LIN {X 0,Y 267.437,Z 177.913,A -85,B 0,C 180,E1 11882.304,E2 11882.304} C_VEL
LIN {X 0,Y 262.666,Z 169.182,A -85,B 0,C 180,E1 11878.91,E2 11878.91} C_VEL
LIN {X 0,Y 261.698,Z 164.317,A -85,B 0,C 180,E1 11875.398,E2 11875.398} C_VEL
LIN {X 0,Y 260.906,Z 160.303,A -85,B 0,C 180,E1 11871.391,E2 11871.391} C_VEL
LIN {X 0,Y 260.574,Z 157.948,A -85,B 0,C 180,E1 11867.817,E2 11867.817} C_VEL
LIN {X 0,Y 260.431,Z 157.03,A -85,B 0,C 180,E1 11862.806,E2 11862.806} C_VEL
LIN {X 0,Y 260.984,Z 157.956,A -85,B 0,C 180,E1 11858.587,E2 11858.587} C_VEL
LIN {X 0,Y 261.9,Z 159.655,A -85,B 0,C 180,E1 11855.41,E2 11855.41} C_VEL
LIN {X 0,Y 263.162,Z 163.319,A -85,B 0,C 180,E1 11851.646,E2 11851.646} C_VEL
LIN {X 0,Y 264.344,Z 166.629,A -85,B 0,C 180,E1 11849.225,E2 11849.225} C_VEL
LIN {X 0,Y 269.556,Z 174.246,A -85,B 0,C 180,E1 11846.002,E2 11846.002} C_VEL
LIN {X 0,Y 274.151,Z 181.59,A -85,B 0,C 180,E1 11843.655,E2 11843.655} C_VEL
LIN {X 0,Y 279.034,Z 190.083,A -85,B 0,C 180,E1 11841.462,E2 11841.462} C_VEL
LIN {X 0,Y 281.087,Z 194.443,A -85,B 0,C 180,E1 11840.571,E2 11840.571} C_VEL
LIN {X 0,Y 281.207,Z 206.246,A -85,B 0,C 180,E1 11839.931,E2 11839.931} C_VEL
LIN {X 0,Y 271.188,Z 340.936,A -85,B 0,C 180,E1 11836.322,E2 11836.322} C_VEL
LIN {X 0,Y 268.525,Z 359.447,A -85,B 0,C 180,E1 11835.523,E2 11835.523} C_VEL
LIN {X 0,Y 264.865,Z 376.74,A -85,B 0,C 180,E1 11834.449,E2 11834.449} C_VEL
LIN {X 0,Y 260.399,Z 393.338,A -85,B 0,C 180,E1 11833.028,E2 11833.028} C_VEL
LIN {X 0,Y 255.563,Z 408.467,A -85,B 0,C 180,E1 11831.308,E2 11831.308} C_VEL
LIN {X 0,Y 250.235,Z 423.172,A -85,B 0,C 180,E1 11829.149,E2 11829.149} C_VEL
LIN {X 0,Y 244.431,Z 437.876,A -85,B 0,C 180,E1 11826.381,E2 11826.381} C_VEL
LIN {X 0,Y 238.982,Z 450.923,A -85,B 0,C 180,E1 11823.237,E2 11823.237} C_VEL
LIN {X 0,Y 234.103,Z 462.435,A -85,B 0,C 180,E1 11819.7,E2 11819.7} C_VEL
LIN {X 0,Y 230.027,Z 472.48,A -85,B 0,C 180,E1 11815.766,E2 11815.766} C_VEL
LIN {X 0,Y 226.993,Z 481.069,A -85,B 0,C 180,E1 11811.446,E2 11811.446} C_VEL
LIN {X 0,Y 225.186,Z 488.132,A -85,B 0,C 180,E1 11806.776,E2 11806.776} C_VEL
LIN {X 0,Y 224.728,Z 493.306,A -85,B 0,C 180,E1 11802.072,E2 11802.072} C_VEL
LIN {X 0,Y 225.341,Z 496.657,A -85,B 0,C 180,E1 11797.395,E2 11797.395} C_VEL
LIN {X 0,Y 226.348,Z 498.067,A -85,B 0,C 180,E1 11793.294,E2 11793.294} C_VEL
LIN {X 0,Y 226.857,Z 498.055,A -85,B 0,C 180,E1 11790.002,E2 11790.002} C_VEL
LIN {X 0,Y 226.415,Z 496.907,A -85,B 0,C 180,E1 11786.394,E2 11786.394} C_VEL
LIN {X 0,Y 225.507,Z 494.955,A -85,B 0,C 180,E1 11782.614,E2 11782.614} C_VEL
LIN {X 0,Y 224.98,Z 491.385,A -85,B 0,C 180,E1 11778.985,E2 11778.985} C_VEL
LIN {X 0,Y 225.066,Z 485.569,A -85,B 0,C 180,E1 11775.071,E2 11775.071} C_VEL
LIN {X 0,Y 225.901,Z 477.705,A -85,B 0,C 180,E1 11771.294,E2 11771.294} C_VEL
LIN {X 0,Y 228.497,Z 464.106,A -85,B 0,C 180,E1 11765.989,E2 11765.989} C_VEL
LIN {X 0,Y 231.379,Z 452.377,A -85,B 0,C 180,E1 11762.358,E2 11762.358} C_VEL
LIN {X 0,Y 234.793,Z 439.326,A -85,B 0,C 180,E1 11759.129,E2 11759.129} C_VEL
LIN {X 0,Y 238.397,Z 425.351,A -85,B 0,C 180,E1 11756.387,E2 11756.387} C_VEL
LIN {X 0,Y 242.028,Z 410.421,A -85,B 0,C 180,E1 11754.067,E2 11754.067} C_VEL
LIN {X 0,Y 245.616,Z 393.93,A -85,B 0,C 180,E1 11752.073,E2 11752.073} C_VEL
LIN {X 0,Y 248.682,Z 377.423,A -85,B 0,C 180,E1 11750.564,E2 11750.564} C_VEL
LIN {X 0,Y 251.306,Z 359.444,A -85,B 0,C 180,E1 11749.376,E2 11749.376} C_VEL
LIN {X 0,Y 252.921,Z 341.212,A -85,B 0,C 180,E1 11748.58,E2 11748.58} C_VEL
LIN {X 0,Y 260.465,Z 182.567,A -85,B 0,C 180,E1 11744.28,E2 11744.28} C_VEL
LIN {X 0,Y 260.223,Z 166.645,A -85,B 0,C 180,E1 11743.682,E2 11743.682} C_VEL
LIN {X 0,Y 256.691,Z 159.312,A -85,B 0,C 180,E1 11742.821,E2 11742.821} C_VEL
LIN {X 0,Y 249.435,Z 140.807,A -85,B 0,C 180,E1 11739.148,E2 11739.148} C_VEL
LIN {X 0,Y 242.573,Z 125.136,A -85,B 0,C 180,E1 11735.534,E2 11735.534} C_VEL
LIN {X 0,Y 235.678,Z 110.896,A -85,B 0,C 180,E1 11731.74,E2 11731.74} C_VEL
LIN {X 0,Y 230.937,Z 101.989,A -85,B 0,C 180,E1 11729.006,E2 11729.006} C_VEL
LIN {X 0,Y 229.132,Z 98.21,A -85,B 0,C 180,E1 11727.834,E2 11727.834} C_VEL
LIN {X 0,Y 227.177,Z 95.014,A -85,B 0,C 180,E1 11726.674,E2 11726.674} C_VEL
LIN {X 0,Y 226.869,Z 93.749,A -85,B 0,C 180,E1 11726.149,E2 11726.149} C_VEL
LIN {X 0,Y 226.849,Z 93.536,A -85,B 0,C 180,E1 11720.875,E2 11720.875} C_VEL
LIN {X 0,Y 226.834,Z 93.529,A -85,B 0,C 180,E1 11715.597,E2 11715.597} C_VEL
LIN {X 0,Y 226.832,Z 93.525,A -85,B 0,C 180,E1 11710.411,E2 11710.411} C_VEL
LIN {X 0,Y 226.837,Z 93.521,A -85,B 0,C 180,E1 11705.311,E2 11705.311} C_VEL
LIN {X 0,Y 226.825,Z 93.521,A -85,B 0,C 180,E1 11699.999,E2 11699.999} C_VEL
LIN {X 0,Y 226.83,Z 93.523,A -85,B 0,C 180,E1 11694.942,E2 11694.942} C_VEL
LIN {X 0,Y 226.833,Z 93.526,A -85,B 0,C 180,E1 11689.587,E2 11689.587} C_VEL
LIN {X 0,Y 226.866,Z 93.724,A -85,B 0,C 180,E1 11685.711,E2 11685.711} C_VEL
LIN {X 0,Y 227.21,Z 95.191,A -85,B 0,C 180,E1 11684.69,E2 11684.69} C_VEL
LIN {X 0,Y 229.356,Z 98.44,A -85,B 0,C 180,E1 11682.494,E2 11682.494} C_VEL
LIN {X 0,Y 230.666,Z 99.715,A -85,B 0,C 180,E1 11681.421,E2 11681.421} C_VEL
LIN {X 0,Y 232.401,Z 103.285,A -85,B 0,C 180,E1 11679.605,E2 11679.605} C_VEL
LIN {X 0,Y 233.957,Z 105.019,A -85,B 0,C 180,E1 11678.436,E2 11678.436} C_VEL
LIN {X 0,Y 236.12,Z 109.062,A -85,B 0,C 180,E1 11676.543,E2 11676.543} C_VEL
LIN {X 0,Y 237.292,Z 111.038,A -85,B 0,C 180,E1 11675.61,E2 11675.61} C_VEL
LIN {X 0,Y 240.213,Z 116.403,A -85,B 0,C 180,E1 11673.285,E2 11673.285} C_VEL
LIN {X 0,Y 243.943,Z 123.406,A -85,B 0,C 180,E1 11670.537,E2 11670.537} C_VEL
LIN {X 0,Y 248.961,Z 134.345,A -85,B 0,C 180,E1 11666.893,E2 11666.893} C_VEL
LIN {X 0,Y 253.489,Z 146.18,A -85,B 0,C 180,E1 11663.444,E2 11663.444} C_VEL
LIN {X 0,Y 257.748,Z 159.766,A -85,B 0,C 180,E1 11660.057,E2 11660.057} C_VEL
LIN {X 0,Y 259.774,Z 168.609,A -85,B 0,C 180,E1 11658.136,E2 11658.136} C_VEL
LIN {X 0,Y 256.196,Z 205.517,A -85,B 0,C 180,E1 11653.073,E2 11653.073} C_VEL
LIN {X 0,Y 255.073,Z 219.925,A -85,B 0,C 180,E1 11651.192,E2 11651.192} C_VEL
LIN {X 0,Y 255.745,Z 226.346,A -85,B 0,C 180,E1 11650.844,E2 11650.844} C_VEL
LIN {X 0,Y 251.79,Z 315.486,A -85,B 0,C 180,E1 11648.415,E2 11648.415} C_VEL
LIN {X 0,Y 251.344,Z 337.034,A -85,B 0,C 180,E1 11647.632,E2 11647.632} C_VEL
LIN {X 0,Y 250.337,Z 351.44,A -85,B 0,C 180,E1 11646.724,E2 11646.724} C_VEL
LIN {X 0,Y 248.542,Z 365.675,A -85,B 0,C 180,E1 11645.398,E2 11645.398} C_VEL
LIN {X 0,Y 246.267,Z 378.333,A -85,B 0,C 180,E1 11643.793,E2 11643.793} C_VEL
LIN {X 0,Y 243.611,Z 390.139,A -85,B 0,C 180,E1 11641.831,E2 11641.831} C_VEL
LIN {X 0,Y 240.515,Z 401.442,A -85,B 0,C 180,E1 11639.374,E2 11639.374} C_VEL
LIN {X 0,Y 237.305,Z 411.378,A -85,B 0,C 180,E1 11636.524,E2 11636.524} C_VEL
LIN {X 0,Y 234.397,Z 419.352,A -85,B 0,C 180,E1 11633.49,E2 11633.49} C_VEL
LIN {X 0,Y 231.822,Z 425.764,A -85,B 0,C 180,E1 11630.182,E2 11630.182} C_VEL
LIN {X 0,Y 229.746,Z 430.445,A -85,B 0,C 180,E1 11626.69,E2 11626.69} C_VEL
LIN {X 0,Y 228.185,Z 433.478,A -85,B 0,C 180,E1 11622.911,E2 11622.911} C_VEL
LIN {X 0,Y 227.257,Z 434.673,A -85,B 0,C 180,E1 11619.111,E2 11619.111} C_VEL
LIN {X 0,Y 226.912,Z 434.059,A -85,B 0,C 180,E1 11615.219,E2 11615.219} C_VEL
LIN {X 0,Y 227.15,Z 431.504,A -85,B 0,C 180,E1 11611.259,E2 11611.259} C_VEL
LIN {X 0,Y 227.948,Z 427.101,A -85,B 0,C 180,E1 11607.484,E2 11607.484} C_VEL
LIN {X 0,Y 229.216,Z 421.057,A -85,B 0,C 180,E1 11603.989,E2 11603.989} C_VEL
LIN {X 0,Y 230.876,Z 413.508,A -85,B 0,C 180,E1 11600.778,E2 11600.778} C_VEL
LIN {X 0,Y 232.823,Z 404.48,A -85,B 0,C 180,E1 11597.851,E2 11597.851} C_VEL
LIN {X 0,Y 235.023,Z 393.302,A -85,B 0,C 180,E1 11595.083,E2 11595.083} C_VEL
LIN {X 0,Y 236.437,Z 385.836,A -85,B 0,C 180,E1 11593.539,E2 11593.539} C_VEL
LIN {X 0,Y 237.322,Z 385.675,A -85,B 0,C 180,E1 11593.098,E2 11593.098} C_VEL
LIN {X 0,Y 237.457,Z 386.342,A -85,B 0,C 180,E1 11592.909,E2 11592.909} C_VEL
LIN {X 0,Y 234.65,Z 398.324,A -85,B 0,C 180,E1 11590.068,E2 11590.068} C_VEL
LIN {X 0,Y 232.114,Z 408.776,A -85,B 0,C 180,E1 11586.92,E2 11586.92} C_VEL
LIN {X 0,Y 229.927,Z 417.813,A -85,B 0,C 180,E1 11583.389,E2 11583.389} C_VEL
LIN {X 0,Y 228.359,Z 424.842,A -85,B 0,C 180,E1 11579.765,E2 11579.765} C_VEL
LIN {X 0,Y 227.33,Z 430.447,A -85,B 0,C 180,E1 11575.736,E2 11575.736} C_VEL
LIN {X 0,Y 226.986,Z 433.918,A -85,B 0,C 180,E1 11571.923,E2 11571.923} C_VEL
LIN {X 0,Y 227.285,Z 435.822,A -85,B 0,C 180,E1 11567.694,E2 11567.694} C_VEL
LIN {X 0,Y 228.271,Z 435.874,A -85,B 0,C 180,E1 11563.719,E2 11563.719} C_VEL
LIN {X 0,Y 230.027,Z 434.082,A -85,B 0,C 180,E1 11559.701,E2 11559.701} C_VEL
LIN {X 0,Y 232.613,Z 430.513,A -85,B 0,C 180,E1 11555.774,E2 11555.774} C_VEL
LIN {X 0,Y 235.937,Z 425.091,A -85,B 0,C 180,E1 11552.05,E2 11552.05} C_VEL
LIN {X 0,Y 240.029,Z 417.755,A -85,B 0,C 180,E1 11548.484,E2 11548.484} C_VEL
LIN {X 0,Y 244.454,Z 408.927,A -85,B 0,C 180,E1 11545.319,E2 11545.319} C_VEL
LIN {X 0,Y 249.258,Z 398.306,A -85,B 0,C 180,E1 11542.401,E2 11542.401} C_VEL
LIN {X 0,Y 253.856,Z 386.726,A -85,B 0,C 180,E1 11539.953,E2 11539.953} C_VEL
LIN {X 0,Y 258.341,Z 373.716,A -85,B 0,C 180,E1 11537.804,E2 11537.804} C_VEL
LIN {X 0,Y 262.44,Z 359.675,A -85,B 0,C 180,E1 11535.998,E2 11535.998} C_VEL
LIN {X 0,Y 266.113,Z 344.035,A -85,B 0,C 180,E1 11534.47,E2 11534.47} C_VEL
LIN {X 0,Y 268.945,Z 328.005,A -85,B 0,C 180,E1 11533.321,E2 11533.321} C_VEL
LIN {X 0,Y 271.021,Z 310.302,A -85,B 0,C 180,E1 11532.464,E2 11532.464} C_VEL
LIN {X 0,Y 273.763,Z 280.354,A -85,B 0,C 180,E1 11531.473,E2 11531.473} C_VEL
LIN {X 0,Y 273.908,Z 272.836,A -85,B 0,C 180,E1 11531.068,E2 11531.068} C_VEL
LIN {X 0,Y 272.225,Z 253.256,A -85,B 0,C 180,E1 11529.371,E2 11529.371} C_VEL
LIN {X 0,Y 272.444,Z 246.79,A -85,B 0,C 180,E1 11529.038,E2 11529.038} C_VEL
LIN {X 0,Y 273.723,Z 232.593,A -85,B 0,C 180,E1 11528.561,E2 11528.561} C_VEL
LIN {X 0,Y 272.08,Z 208.308,A -85,B 0,C 180,E1 11526.436,E2 11526.436} C_VEL
LIN {X 0,Y 271.119,Z 198.139,A -85,B 0,C 180,E1 11525.371,E2 11525.371} C_VEL
LIN {X 0,Y 267.119,Z 189.254,A -85,B 0,C 180,E1 11523.058,E2 11523.058} C_VEL
LIN {X 0,Y 263.16,Z 181.691,A -85,B 0,C 180,E1 11520.49,E2 11520.49} C_VEL
LIN {X 0,Y 259.632,Z 175.218,A -85,B 0,C 180,E1 11517.738,E2 11517.738} C_VEL
LIN {X 0,Y 256.045,Z 168.731,A -85,B 0,C 180,E1 11513.948,E2 11513.948} C_VEL
LIN {X 0,Y 255.481,Z 165.908,A -85,B 0,C 180,E1 11510.767,E2 11510.767} C_VEL
LIN {X 0,Y 255.299,Z 163.935,A -85,B 0,C 180,E1 11507.561,E2 11507.561} C_VEL
LIN {X 0,Y 255.269,Z 163.135,A -85,B 0,C 180,E1 11502.682,E2 11502.682} C_VEL
LIN {X 0,Y 255.846,Z 164.125,A -85,B 0,C 180,E1 11498.448,E2 11498.448} C_VEL
LIN {X 0,Y 256.662,Z 165.634,A -85,B 0,C 180,E1 11495.611,E2 11495.611} C_VEL
LIN {X 0,Y 257.557,Z 167.784,A -85,B 0,C 180,E1 11493.609,E2 11493.609} C_VEL
LIN {X 0,Y 261.58,Z 173.047,A -85,B 0,C 180,E1 11490.192,E2 11490.192} C_VEL
LIN {X 0,Y 267.003,Z 181.165,A -85,B 0,C 180,E1 11486.665,E2 11486.665} C_VEL
LIN {X 0,Y 271.33,Z 188.369,A -85,B 0,C 180,E1 11484.328,E2 11484.328} C_VEL
LIN {X 0,Y 275.963,Z 196.912,A -85,B 0,C 180,E1 11482.112,E2 11482.112} C_VEL
LIN {X 0,Y 276.768,Z 198.93,A -85,B 0,C 180,E1 11481.73,E2 11481.73} C_VEL
LIN {X 0,Y 276.718,Z 207.567,A -85,B 0,C 180,E1 11481.275,E2 11481.275} C_VEL
LIN {X 0,Y 266.246,Z 340.353,A -85,B 0,C 180,E1 11477.677,E2 11477.677} C_VEL
LIN {X 0,Y 263.401,Z 359.063,A -85,B 0,C 180,E1 11476.859,E2 11476.859} C_VEL
LIN {X 0,Y 259.545,Z 376.363,A -85,B 0,C 180,E1 11475.771,E2 11475.771} C_VEL
LIN {X 0,Y 254.777,Z 393.099,A -85,B 0,C 180,E1 11474.312,E2 11474.312} C_VEL
LIN {X 0,Y 249.474,Z 408.834,A -85,B 0,C 180,E1 11472.486,E2 11472.486} C_VEL
LIN {X 0,Y 243.534,Z 424.298,A -85,B 0,C 180,E1 11470.136,E2 11470.136} C_VEL
LIN {X 0,Y 237.723,Z 438.078,A -85,B 0,C 180,E1 11467.429,E2 11467.429} C_VEL
LIN {X 0,Y 232.198,Z 450.45,A -85,B 0,C 180,E1 11464.341,E2 11464.341} C_VEL
LIN {X 0,Y 227.018,Z 461.815,A -85,B 0,C 180,E1 11460.725,E2 11460.725} C_VEL
LIN {X 0,Y 222.615,Z 471.818,A -85,B 0,C 180,E1 11456.647,E2 11456.647} C_VEL
LIN {X 0,Y 219.2,Z 480.673,A -85,B 0,C 180,E1 11451.966,E2 11451.966} C_VEL
LIN {X 0,Y 217.26,Z 487.562,A -85,B 0,C 180,E1 11447.132,E2 11447.132} C_VEL
LIN {X 0,Y 216.746,Z 492.532,A -85,B 0,C 180,E1 11442.253,E2 11442.253} C_VEL
LIN {X 0,Y 217.378,Z 495.68,A -85,B 0,C 180,E1 11437.402,E2 11437.402} C_VEL
LIN {X 0,Y 218.442,Z 496.977,A -85,B 0,C 180,E1 11433.151,E2 11433.151} C_VEL
LIN {X 0,Y 218.941,Z 496.809,A -85,B 0,C 180,E1 11429.74,E2 11429.74} C_VEL
LIN {X 0,Y 218.377,Z 495.767,A -85,B 0,C 180,E1 11426.064,E2 11426.064} C_VEL
LIN {X 0,Y 217.42,Z 493.706,A -85,B 0,C 180,E1 11422.072,E2 11422.072} C_VEL
LIN {X 0,Y 216.956,Z 490.038,A -85,B 0,C 180,E1 11418.303,E2 11418.303} C_VEL
LIN {X 0,Y 217.131,Z 484.595,A -85,B 0,C 180,E1 11414.512,E2 11414.512} C_VEL
LIN {X 0,Y 218.066,Z 477.076,A -85,B 0,C 180,E1 11410.726,E2 11410.726} C_VEL
LIN {X 0,Y 219.647,Z 467.956,A -85,B 0,C 180,E1 11407.239,E2 11407.239} C_VEL
LIN {X 0,Y 222.595,Z 455.787,A -85,B 0,C 180,E1 11403.023,E2 11403.023} C_VEL
LIN {X 0,Y 225.976,Z 443.237,A -85,B 0,C 180,E1 11399.564,E2 11399.564} C_VEL
LIN {X 0,Y 229.664,Z 429.655,A -85,B 0,C 180,E1 11396.586,E2 11396.586} C_VEL
LIN {X 0,Y 233.602,Z 414.453,A -85,B 0,C 180,E1 11393.951,E2 11393.951} C_VEL
LIN {X 0,Y 237.23,Z 399.105,A -85,B 0,C 180,E1 11391.872,E2 11391.872} C_VEL
LIN {X 0,Y 240.529,Z 383.043,A -85,B 0,C 180,E1 11390.199,E2 11390.199} C_VEL
LIN {X 0,Y 243.443,Z 365.595,A -85,B 0,C 180,E1 11388.866,E2 11388.866} C_VEL
LIN {X 0,Y 245.477,Z 347.732,A -85,B 0,C 180,E1 11387.924,E2 11387.924} C_VEL
LIN {X 0,Y 246.866,Z 323.354,A -85,B 0,C 180,E1 11387.15,E2 11387.15} C_VEL
LIN {X 0,Y 253.844,Z 182.685,A -85,B 0,C 180,E1 11383.269,E2 11383.269} C_VEL
LIN {X 0,Y 253.611,Z 169.351,A -85,B 0,C 180,E1 11382.75,E2 11382.75} C_VEL
LIN {X 0,Y 248.793,Z 159.479,A -85,B 0,C 180,E1 11381.537,E2 11381.537} C_VEL
LIN {X 0,Y 241.466,Z 141.002,A -85,B 0,C 180,E1 11377.644,E2 11377.644} C_VEL
LIN {X 0,Y 233.932,Z 124.103,A -85,B 0,C 180,E1 11373.46,E2 11373.46} C_VEL
LIN {X 0,Y 227.609,Z 111.471,A -85,B 0,C 180,E1 11369.761,E2 11369.761} C_VEL
LIN {X 0,Y 223.929,Z 104.042,A -85,B 0,C 180,E1 11367.315,E2 11367.315} C_VEL
LIN {X 0,Y 222.712,Z 100.733,A -85,B 0,C 180,E1 11365.815,E2 11365.815} C_VEL
LIN {X 0,Y 219.505,Z 96.717,A -85,B 0,C 180,E1 11362.214,E2 11362.214} C_VEL
LIN {X 0,Y 218.978,Z 94.969,A -85,B 0,C 180,E1 11360.863,E2 11360.863} C_VEL
LIN {X 0,Y 218.897,Z 94.512,A -85,B 0,C 180,E1 11358.371,E2 11358.371} C_VEL
LIN {X 0,Y 218.904,Z 94.517,A -85,B 0,C 180,E1 11352.932,E2 11352.932} C_VEL
LIN {X 0,Y 218.909,Z 94.525,A -85,B 0,C 180,E1 11347.347,E2 11347.347} C_VEL
LIN {X 0,Y 218.891,Z 94.526,A -85,B 0,C 180,E1 11341.832,E2 11341.832} C_VEL
LIN {X 0,Y 218.887,Z 94.522,A -85,B 0,C 180,E1 11336.595,E2 11336.595} C_VEL
LIN {X 0,Y 218.917,Z 94.71,A -85,B 0,C 180,E1 11331.86,E2 11331.86} C_VEL
LIN {X 0,Y 219.316,Z 96.294,A -85,B 0,C 180,E1 11330.288,E2 11330.288} C_VEL
LIN {X 0,Y 221.6,Z 99.581,A -85,B 0,C 180,E1 11327.226,E2 11327.226} C_VEL
LIN {X 0,Y 223.03,Z 100.894,A -85,B 0,C 180,E1 11325.725,E2 11325.725} C_VEL
LIN {X 0,Y 224.788,Z 104.559,A -85,B 0,C 180,E1 11323.46,E2 11323.46} C_VEL
LIN {X 0,Y 226.477,Z 106.174,A -85,B 0,C 180,E1 11321.998,E2 11321.998} C_VEL
LIN {X 0,Y 228.612,Z 110.328,A -85,B 0,C 180,E1 11319.786,E2 11319.786} C_VEL
LIN {X 0,Y 229.8,Z 111.833,A -85,B 0,C 180,E1 11318.83,E2 11318.83} C_VEL
LIN {X 0,Y 232.256,Z 116.102,A -85,B 0,C 180,E1 11316.667,E2 11316.667} C_VEL
LIN {X 0,Y 235.578,Z 122.558,A -85,B 0,C 180,E1 11313.806,E2 11313.806} C_VEL
LIN {X 0,Y 239.434,Z 130.272,A -85,B 0,C 180,E1 11310.752,E2 11310.752} C_VEL
LIN {X 0,Y 243.738,Z 139.831,A -85,B 0,C 180,E1 11307.493,E2 11307.493} C_VEL
LIN {X 0,Y 248.092,Z 151.68,A -85,B 0,C 180,E1 11303.955,E2 11303.955} C_VEL
LIN {X 0,Y 252.159,Z 165.376,A -85,B 0,C 180,E1 11300.474,E2 11300.474} C_VEL
LIN {X 0,Y 253.596,Z 172.022,A -85,B 0,C 180,E1 11299.025,E2 11299.025} C_VEL
LIN {X 0,Y 249.713,Z 209.361,A -85,B 0,C 180,E1 11293.841,E2 11293.841} C_VEL
LIN {X 0,Y 248.794,Z 220.984,A -85,B 0,C 180,E1 11292.325,E2 11292.325} C_VEL
LIN {X 0,Y 249.464,Z 227.522,A -85,B 0,C 180,E1 11291.955,E2 11291.955} C_VEL
LIN {X 0,Y 245.334,Z 315.798,A -85,B 0,C 180,E1 11289.503,E2 11289.503} C_VEL
LIN {X 0,Y 244.824,Z 338.009,A -85,B 0,C 180,E1 11288.681,E2 11288.681} C_VEL
LIN {X 0,Y 243.717,Z 352.801,A -85,B 0,C 180,E1 11287.725,E2 11287.725} C_VEL
LIN {X 0,Y 241.845,Z 366.822,A -85,B 0,C 180,E1 11286.386,E2 11286.386} C_VEL
LIN {X 0,Y 239.454,Z 379.469,A -85,B 0,C 180,E1 11284.745,E2 11284.745} C_VEL
LIN {X 0,Y 236.657,Z 391.281,A -85,B 0,C 180,E1 11282.735,E2 11282.735} C_VEL
LIN {X 0,Y 233.551,Z 402.077,A -85,B 0,C 180,E1 11280.34,E2 11280.34} C_VEL
LIN {X 0,Y 230.422,Z 411.382,A -85,B 0,C 180,E1 11277.662,E2 11277.662} C_VEL
LIN {X 0,Y 227.423,Z 419.334,A -85,B 0,C 180,E1 11274.685,E2 11274.685} C_VEL
LIN {X 0,Y 224.504,Z 426.271,A -85,B 0,C 180,E1 11271.143,E2 11271.143} C_VEL
LIN {X 0,Y 222.157,Z 431.261,A -85,B 0,C 180,E1 11267.416,E2 11267.416} C_VEL
LIN {X 0,Y 220.488,Z 434.358,A -85,B 0,C 180,E1 11263.637,E2 11263.637} C_VEL
LIN {X 0,Y 219.434,Z 435.746,A -85,B 0,C 180,E1 11259.704,E2 11259.704} C_VEL
LIN {X 0,Y 218.989,Z 435.247,A -85,B 0,C 180,E1 11255.5,E2 11255.5} C_VEL
LIN {X 0,Y 219.211,Z 432.705,A -85,B 0,C 180,E1 11251.305,E2 11251.305} C_VEL
LIN {X 0,Y 220.029,Z 428.354,A -85,B 0,C 180,E1 11247.394,E2 11247.394} C_VEL
LIN {X 0,Y 221.346,Z 422.381,A -85,B 0,C 180,E1 11243.774,E2 11243.774} C_VEL
LIN {X 0,Y 223.077,Z 414.913,A -85,B 0,C 180,E1 11240.452,E2 11240.452} C_VEL
LIN {X 0,Y 225.107,Z 405.961,A -85,B 0,C 180,E1 11237.428,E2 11237.428} C_VEL
LIN {X 0,Y 227.407,Z 394.888,A -85,B 0,C 180,E1 11234.572,E2 11234.572} C_VEL
LIN {X 0,Y 228.503,Z 389.806,A -85,B 0,C 180,E1 11233.409,E2 11233.409} C_VEL
LIN {X 0,Y 229.328,Z 389.886,A -85,B 0,C 180,E1 11232.971,E2 11232.971} C_VEL
LIN {X 0,Y 226.535,Z 401.239,A -85,B 0,C 180,E1 11230.073,E2 11230.073} C_VEL
LIN {X 0,Y 223.811,Z 411.913,A -85,B 0,C 180,E1 11226.57,E2 11226.57} C_VEL
LIN {X 0,Y 221.82,Z 419.934,A -85,B 0,C 180,E1 11223.189,E2 11223.189} C_VEL
LIN {X 0,Y 220.28,Z 426.66,A -85,B 0,C 180,E1 11219.443,E2 11219.443} C_VEL
LIN {X 0,Y 219.361,Z 431.736,A -85,B 0,C 180,E1 11215.582,E2 11215.582} C_VEL
LIN {X 0,Y 219.047,Z 435.139,A -85,B 0,C 180,E1 11211.625,E2 11211.625} C_VEL
LIN {X 0,Y 219.443,Z 437.024,A -85,B 0,C 180,E1 11207.188,E2 11207.188} C_VEL
LIN {X 0,Y 220.545,Z 437.016,A -85,B 0,C 180,E1 11203.12,E2 11203.12} C_VEL
LIN {X 0,Y 222.483,Z 435.207,A -85,B 0,C 180,E1 11198.968,E2 11198.968} C_VEL
LIN {X 0,Y 225.293,Z 431.623,A -85,B 0,C 180,E1 11194.926,E2 11194.926} C_VEL
LIN {X 0,Y 228.959,Z 426.06,A -85,B 0,C 180,E1 11191.018,E2 11191.018} C_VEL
LIN {X 0,Y 233.245,Z 418.921,A -85,B 0,C 180,E1 11187.455,E2 11187.455} C_VEL
LIN {X 0,Y 237.935,Z 410.138,A -85,B 0,C 180,E1 11184.231,E2 11184.231} C_VEL
LIN {X 0,Y 243.083,Z 399.386,A -85,B 0,C 180,E1 11181.222,E2 11181.222} C_VEL
LIN {X 0,Y 248.05,Z 387.616,A -85,B 0,C 180,E1 11178.689,E2 11178.689} C_VEL
LIN {X 0,Y 253.07,Z 373.858,A -85,B 0,C 180,E1 11176.398,E2 11176.398} C_VEL
LIN {X 0,Y 257.292,Z 359.881,A -85,B 0,C 180,E1 11174.614,E2 11174.614} C_VEL
LIN {X 0,Y 261.218,Z 343.765,A -85,B 0,C 180,E1 11173.052,E2 11173.052} C_VEL
LIN {X 0,Y 264.173,Z 327.239,A -85,B 0,C 180,E1 11171.898,E2 11171.898} C_VEL
LIN {X 0,Y 266.246,Z 310.037,A -85,B 0,C 180,E1 11171.08,E2 11171.08} C_VEL
LIN {X 0,Y 272.444,Z 246.79,A -85,B 0,C 180,E1 11169.038,E2 11169.038} C_VEL
LIN {X 0,Y 272.523,Z 240.406,A -85,B 0,C 180,E1 11168.661,E2 11168.661} C_VEL
LIN {X 0,Y 271.427,Z 232.549,A -85,B 0,C 180,E1 11167.79,E2 11167.79} C_VEL
LIN {X 0,Y 268.628,Z 218.323,A -85,B 0,C 180,E1 11165.829,E2 11165.829} C_VEL
LIN {X 0,Y 268.341,Z 215.259,A -85,B 0,C 180,E1 11165.502,E2 11165.502} C_VEL
LIN {X 0,Y 267.385,Z 203.08,A -85,B 0,C 180,E1 11164.236,E2 11164.236} C_VEL
LIN {X 0,Y 263.628,Z 194.556,A -85,B 0,C 180,E1 11161.848,E2 11161.848} C_VEL
LIN {X 0,Y 260.658,Z 188.463,A -85,B 0,C 180,E1 11159.726,E2 11159.726} C_VEL
LIN {X 0,Y 257.518,Z 182.41,A -85,B 0,C 180,E1 11157.107,E2 11157.107} C_VEL
LIN {X 0,Y 254.087,Z 176.087,A -85,B 0,C 180,E1 11153.334,E2 11153.334} C_VEL
LIN {X 0,Y 252.12,Z 172.886,A -85,B 0,C 180,E1 11150.182,E2 11150.182} C_VEL
LIN {X 0,Y 251.149,Z 170.743,A -85,B 0,C 180,E1 11147.352,E2 11147.352} C_VEL
LIN {X 0,Y 250.991,Z 169.905,A -85,B 0,C 180,E1 11142.855,E2 11142.855} C_VEL
LIN {X 0,Y 252.188,Z 171.067,A -85,B 0,C 180,E1 11139.095,E2 11139.095} C_VEL
LIN {X 0,Y 254.355,Z 173.288,A -85,B 0,C 180,E1 11135.782,E2 11135.782} C_VEL
LIN {X 0,Y 257.471,Z 177.622,A -85,B 0,C 180,E1 11132.476,E2 11132.476} C_VEL
LIN {X 0,Y 260.529,Z 181.918,A -85,B 0,C 180,E1 11130.009,E2 11130.009} C_VEL
LIN {X 0,Y 264.676,Z 188.384,A -85,B 0,C 180,E1 11127.238,E2 11127.238} C_VEL
LIN {X 0,Y 268.619,Z 195.289,A -85,B 0,C 180,E1 11124.975,E2 11124.975} C_VEL
LIN {X 0,Y 272.552,Z 203.113,A -85,B 0,C 180,E1 11122.947,E2 11122.947} C_VEL
LIN {X 0,Y 272.362,Z 209.267,A -85,B 0,C 180,E1 11122.652,E2 11122.652} C_VEL
LIN {X 0,Y 261.497,Z 339.487,A -85,B 0,C 180,E1 11119.093,E2 11119.093} C_VEL
LIN {X 0,Y 258.551,Z 358.19,A -85,B 0,C 180,E1 11118.278,E2 11118.278} C_VEL
LIN {X 0,Y 254.571,Z 375.453,A -85,B 0,C 180,E1 11117.197,E2 11117.197} C_VEL
LIN {X 0,Y 249.73,Z 391.838,A -85,B 0,C 180,E1 11115.782,E2 11115.782} C_VEL
LIN {X 0,Y 244.172,Z 407.57,A -85,B 0,C 180,E1 11113.956,E2 11113.956} C_VEL
LIN {X 0,Y 238.195,Z 422.368,A -85,B 0,C 180,E1 11111.709,E2 11111.709} C_VEL
LIN {X 0,Y 232.021,Z 436.297,A -85,B 0,C 180,E1 11108.99,E2 11108.99} C_VEL
LIN {X 0,Y 225.914,Z 449.198,A -85,B 0,C 180,E1 11105.749,E2 11105.749} C_VEL
LIN {X 0,Y 220.347,Z 460.536,A -85,B 0,C 180,E1 11102.068,E2 11102.068} C_VEL
LIN {X 0,Y 215.592,Z 470.475,A -85,B 0,C 180,E1 11097.933,E2 11097.933} C_VEL
LIN {X 0,Y 211.755,Z 479.413,A -85,B 0,C 180,E1 11093.075,E2 11093.075} C_VEL
LIN {X 0,Y 209.497,Z 486.303,A -85,B 0,C 180,E1 11088.075,E2 11088.075} C_VEL
LIN {X 0,Y 208.765,Z 491.297,A -85,B 0,C 180,E1 11083.011,E2 11083.011} C_VEL
LIN {X 0,Y 209.293,Z 494.464,A -85,B 0,C 180,E1 11077.965,E2 11077.965} C_VEL
LIN {X 0,Y 210.405,Z 495.797,A -85,B 0,C 180,E1 11073.544,E2 11073.544} C_VEL
LIN {X 0,Y 211.034,Z 495.667,A -85,B 0,C 180,E1 11070.002,E2 11070.002} C_VEL
LIN {X 0,Y 210.531,Z 494.786,A -85,B 0,C 180,E1 11066.462,E2 11066.462} C_VEL
LIN {X 0,Y 209.553,Z 493.211,A -85,B 0,C 180,E1 11062.6,E2 11062.6} C_VEL
LIN {X 0,Y 208.973,Z 489.656,A -85,B 0,C 180,E1 11058.41,E2 11058.41} C_VEL
LIN {X 0,Y 209.133,Z 484.487,A -85,B 0,C 180,E1 11054.473,E2 11054.473} C_VEL
LIN {X 0,Y 210.003,Z 477.961,A -85,B 0,C 180,E1 11050.824,E2 11050.824} C_VEL
LIN {X 0,Y 211.751,Z 468.663,A -85,B 0,C 180,E1 11046.929,E2 11046.929} C_VEL
LIN {X 0,Y 216.902,Z 447.742,A -85,B 0,C 180,E1 11040.297,E2 11040.297} C_VEL
LIN {X 0,Y 220.799,Z 433.999,A -85,B 0,C 180,E1 11036.902,E2 11036.902} C_VEL
LIN {X 0,Y 224.828,Z 419.401,A -85,B 0,C 180,E1 11034.056,E2 11034.056} C_VEL
LIN {X 0,Y 228.846,Z 403.619,A -85,B 0,C 180,E1 11031.657,E2 11031.657} C_VEL
LIN {X 0,Y 232.391,Z 387.723,A -85,B 0,C 180,E1 11029.81,E2 11029.81} C_VEL
LIN {X 0,Y 235.538,Z 370.803,A -85,B 0,C 180,E1 11028.341,E2 11028.341} C_VEL
LIN {X 0,Y 238.044,Z 352.463,A -85,B 0,C 180,E1 11027.217,E2 11027.217} C_VEL
LIN {X 0,Y 239.454,Z 334.168,A -85,B 0,C 180,E1 11026.496,E2 11026.496} C_VEL
LIN {X 0,Y 247.274,Z 183.883,A -85,B 0,C 180,E1 11022.257,E2 11022.257} C_VEL
LIN {X 0,Y 247.063,Z 172.097,A -85,B 0,C 180,E1 11021.777,E2 11021.777} C_VEL
LIN {X 0,Y 240.942,Z 159.77,A -85,B 0,C 180,E1 11020.187,E2 11020.187} C_VEL
LIN {X 0,Y 234.181,Z 142.771,A -85,B 0,C 180,E1 11016.403,E2 11016.403} C_VEL
LIN {X 0,Y 227.766,Z 128.431,A -85,B 0,C 180,E1 11012.68,E2 11012.68} C_VEL
LIN {X 0,Y 222.97,Z 118.138,A -85,B 0,C 180,E1 11009.553,E2 11009.553} C_VEL
LIN {X 0,Y 220.153,Z 109.945,A -85,B 0,C 180,E1 11006.138,E2 11006.138} C_VEL
LIN {X 0,Y 219.319,Z 107.418,A -85,B 0,C 180,E1 11004.941,E2 11004.941} C_VEL
LIN {X 0,Y 216.571,Z 104.027,A -85,B 0,C 180,E1 11001.817,E2 11001.817} C_VEL
LIN {X 0,Y 215.534,Z 101.862,A -85,B 0,C 180,E1 11000.077,E2 11000.077} C_VEL
LIN {X 0,Y 211.173,Z 96.573,A -85,B 0,C 180,E1 10988.989,E2 10988.989} C_VEL
LIN {X 0,Y 211.11,Z 96.382,A -85,B 0,C 180,E1 10984.345,E2 10984.345} C_VEL
LIN {X 0,Y 211.756,Z 98.105,A -85,B 0,C 180,E1 10979.458,E2 10979.458} C_VEL
LIN {X 0,Y 215.446,Z 102.043,A -85,B 0,C 180,E1 10971.728,E2 10971.728} C_VEL
LIN {X 0,Y 217.646,Z 106.247,A -85,B 0,C 180,E1 10968.069,E2 10968.069} C_VEL
LIN {X 0,Y 219.316,Z 107.672,A -85,B 0,C 180,E1 10966.286,E2 10966.286} C_VEL
LIN {X 0,Y 220.991,Z 111.335,A -85,B 0,C 180,E1 10963.978,E2 10963.978} C_VEL
LIN {X 0,Y 222.788,Z 113.542,A -85,B 0,C 180,E1 10962.23,E2 10962.23} C_VEL
LIN {X 0,Y 225.157,Z 117.72,A -85,B 0,C 180,E1 10959.734,E2 10959.734} C_VEL
LIN {X 0,Y 228.515,Z 123.961,A -85,B 0,C 180,E1 10956.536,E2 10956.536} C_VEL
LIN {X 0,Y 232.438,Z 131.458,A -85,B 0,C 180,E1 10953.148,E2 10953.148} C_VEL
LIN {X 0,Y 237.34,Z 142.425,A -85,B 0,C 180,E1 10949.072,E2 10949.072} C_VEL
LIN {X 0,Y 241.807,Z 154.217,A -85,B 0,C 180,E1 10945.367,E2 10945.367} C_VEL
LIN {X 0,Y 245.626,Z 166.991,A -85,B 0,C 180,E1 10941.923,E2 10941.923} C_VEL
LIN {X 0,Y 247.479,Z 175.454,A -85,B 0,C 180,E1 10939.958,E2 10939.958} C_VEL
LIN {X 0,Y 243.367,Z 212.991,A -85,B 0,C 180,E1 10934.702,E2 10934.702} C_VEL
LIN {X 0,Y 242.619,Z 222.06,A -85,B 0,C 180,E1 10933.515,E2 10933.515} C_VEL
LIN {X 0,Y 243.28,Z 228.746,A -85,B 0,C 180,E1 10933.122,E2 10933.122} C_VEL
LIN {X 0,Y 238.969,Z 316.262,A -85,B 0,C 180,E1 10930.644,E2 10930.644} C_VEL
LIN {X 0,Y 238.385,Z 339.097,A -85,B 0,C 180,E1 10929.781,E2 10929.781} C_VEL
LIN {X 0,Y 237.206,Z 353.907,A -85,B 0,C 180,E1 10928.802,E2 10928.802} C_VEL
LIN {X 0,Y 235.226,Z 367.969,A -85,B 0,C 180,E1 10927.43,E2 10927.43} C_VEL
LIN {X 0,Y 232.711,Z 380.606,A -85,B 0,C 180,E1 10925.753,E2 10925.753} C_VEL
LIN {X 0,Y 229.769,Z 392.41,A -85,B 0,C 180,E1 10923.696,E2 10923.696} C_VEL
LIN {X 0,Y 226.347,Z 403.692,A -85,B 0,C 180,E1 10921.117,E2 10921.117} C_VEL
LIN {X 0,Y 222.786,Z 413.618,A -85,B 0,C 180,E1 10918.112,E2 10918.112} C_VEL
LIN {X 0,Y 219.674,Z 421.279,A -85,B 0,C 180,E1 10915.04,E2 10915.04} C_VEL
LIN {X 0,Y 216.852,Z 427.593,A -85,B 0,C 180,E1 10911.643,E2 10911.643} C_VEL
LIN {X 0,Y 214.309,Z 432.659,A -85,B 0,C 180,E1 10907.651,E2 10907.651} C_VEL
LIN {X 0,Y 212.53,Z 435.683,A -85,B 0,C 180,E1 10903.603,E2 10903.603} C_VEL
LIN {X 0,Y 211.467,Z 436.867,A -85,B 0,C 180,E1 10899.523,E2 10899.523} C_VEL
LIN {X 0,Y 211.058,Z 436.283,A -85,B 0,C 180,E1 10895.435,E2 10895.435} C_VEL
LIN {X 0,Y 211.271,Z 433.895,A -85,B 0,C 180,E1 10891.354,E2 10891.354} C_VEL
LIN {X 0,Y 212.11,Z 429.606,A -85,B 0,C 180,E1 10887.296,E2 10887.296} C_VEL
LIN {X 0,Y 213.363,Z 424.201,A -85,B 0,C 180,E1 10883.811,E2 10883.811} C_VEL
LIN {X 0,Y 215.131,Z 416.963,A -85,B 0,C 180,E1 10880.366,E2 10880.366} C_VEL
LIN {X 0,Y 217.209,Z 408.241,A -85,B 0,C 180,E1 10877.233,E2 10877.233} C_VEL
LIN {X 0,Y 219.479,Z 398.07,A -85,B 0,C 180,E1 10874.407,E2 10874.407} C_VEL
LIN {X 0,Y 220.484,Z 393.799,A -85,B 0,C 180,E1 10873.33,E2 10873.33} C_VEL
LIN {X 0,Y 221.097,Z 393.769,A -85,B 0,C 180,E1 10872.938,E2 10872.938} C_VEL
LIN {X 0,Y 217.866,Z 406.092,A -85,B 0,C 180,E1 10869.429,E2 10869.429} C_VEL
LIN {X 0,Y 215.306,Z 415.71,A -85,B 0,C 180,E1 10865.877,E2 10865.877} C_VEL
LIN {X 0,Y 213.284,Z 423.746,A -85,B 0,C 180,E1 10862.042,E2 10862.042} C_VEL
LIN {X 0,Y 211.927,Z 429.844,A -85,B 0,C 180,E1 10858.1,E2 10858.1} C_VEL
LIN {X 0,Y 211.194,Z 434.608,A -85,B 0,C 180,E1 10853.714,E2 10853.714} C_VEL
LIN {X 0,Y 211.199,Z 437.285,A -85,B 0,C 180,E1 10849.563,E2 10849.563} C_VEL
LIN {X 0,Y 212.01,Z 438.392,A -85,B 0,C 180,E1 10844.973,E2 10844.973} C_VEL
LIN {X 0,Y 213.619,Z 437.63,A -85,B 0,C 180,E1 10840.688,E2 10840.688} C_VEL
LIN {X 0,Y 216.24,Z 434.941,A -85,B 0,C 180,E1 10836.289,E2 10836.289} C_VEL
LIN {X 0,Y 219.51,Z 430.789,A -85,B 0,C 180,E1 10832.394,E2 10832.394} C_VEL
LIN {X 0,Y 223.653,Z 424.683,A -85,B 0,C 180,E1 10828.579,E2 10828.579} C_VEL
LIN {X 0,Y 228.445,Z 416.866,A -85,B 0,C 180,E1 10825.04,E2 10825.04} C_VEL
LIN {X 0,Y 233.592,Z 407.493,A -85,B 0,C 180,E1 10821.864,E2 10821.864} C_VEL
LIN {X 0,Y 238.986,Z 396.416,A -85,B 0,C 180,E1 10818.996,E2 10818.996} C_VEL
LIN {X 0,Y 244.124,Z 384.334,A -85,B 0,C 180,E1 10816.583,E2 10816.583} C_VEL
LIN {X 0,Y 249.442,Z 369.578,A -85,B 0,C 180,E1 10814.323,E2 10814.323} C_VEL
LIN {X 0,Y 253.77,Z 354.983,A -85,B 0,C 180,E1 10812.62,E2 10812.62} C_VEL
LIN {X 0,Y 257.581,Z 338.611,A -85,B 0,C 180,E1 10811.192,E2 10811.192} C_VEL
LIN {X 0,Y 260.276,Z 322.442,A -85,B 0,C 180,E1 10810.187,E2 10810.187} C_VEL
LIN {X 0,Y 262.584,Z 300.666,A -85,B 0,C 180,E1 10809.319,E2 10809.319} C_VEL
LIN {X 0,Y 269.298,Z 234.279,A -85,B 0,C 180,E1 10807.186,E2 10807.186} C_VEL
LIN {X 0,Y 268.341,Z 215.259,A -85,B 0,C 180,E1 10805.502,E2 10805.502} C_VEL
LIN {X 0,Y 267.67,Z 211.699,A -85,B 0,C 180,E1 10804.976,E2 10804.976} C_VEL
LIN {X 0,Y 265.969,Z 208.222,A -85,B 0,C 180,E1 10804.005,E2 10804.005} C_VEL
LIN {X 0,Y 261.424,Z 202.188,A -85,B 0,C 180,E1 10801.412,E2 10801.412} C_VEL
LIN {X 0,Y 258.282,Z 195.368,A -85,B 0,C 180,E1 10799.002,E2 10799.002} C_VEL
LIN {X 0,Y 255.556,Z 189.72,A -85,B 0,C 180,E1 10796.524,E2 10796.524} C_VEL
LIN {X 0,Y 252.446,Z 183.62,A -85,B 0,C 180,E1 10792.833,E2 10792.833} C_VEL
LIN {X 0,Y 250.654,Z 180.476,A -85,B 0,C 180,E1 10789.66,E2 10789.66} C_VEL
LIN {X 0,Y 249.924,Z 178.647,A -85,B 0,C 180,E1 10787.289,E2 10787.289} C_VEL
LIN {X 0,Y 249.764,Z 177.814,A -85,B 0,C 180,E1 10783.009,E2 10783.009} C_VEL
LIN {X 0,Y 250.822,Z 178.825,A -85,B 0,C 180,E1 10779.464,E2 10779.464} C_VEL
LIN {X 0,Y 252.907,Z 181.039,A -85,B 0,C 180,E1 10776.095,E2 10776.095} C_VEL
LIN {X 0,Y 255.764,Z 185.213,A -85,B 0,C 180,E1 10772.908,E2 10772.908} C_VEL
LIN {X 0,Y 258.56,Z 189.335,A -85,B 0,C 180,E1 10770.523,E2 10770.523} C_VEL
LIN {X 0,Y 262.288,Z 195.451,A -85,B 0,C 180,E1 10767.874,E2 10767.874} C_VEL
LIN {X 0,Y 266.257,Z 202.799,A -85,B 0,C 180,E1 10765.456,E2 10765.456} C_VEL
LIN {X 0,Y 268.554,Z 207.687,A -85,B 0,C 180,E1 10764.198,E2 10764.198} C_VEL
LIN {X 0,Y 256.982,Z 339.03,A -85,B 0,C 180,E1 10760.564,E2 10760.564} C_VEL
LIN {X 0,Y 253.881,Z 357.685,A -85,B 0,C 180,E1 10759.746,E2 10759.746} C_VEL
LIN {X 0,Y 249.703,Z 374.947,A -85,B 0,C 180,E1 10758.66,E2 10758.66} C_VEL
LIN {X 0,Y 244.542,Z 391.479,A -85,B 0,C 180,E1 10757.218,E2 10757.218} C_VEL
LIN {X 0,Y 238.761,Z 407.11,A -85,B 0,C 180,E1 10755.392,E2 10755.392} C_VEL
LIN {X 0,Y 232.247,Z 422.438,A -85,B 0,C 180,E1 10753.031,E2 10753.031} C_VEL
LIN {X 0,Y 225.633,Z 436.431,A -85,B 0,C 180,E1 10750.215,E2 10750.215} C_VEL
LIN {X 0,Y 219.352,Z 448.796,A -85,B 0,C 180,E1 10746.993,E2 10746.993} C_VEL
LIN {X 0,Y 213.454,Z 460,A -85,B 0,C 180,E1 10743.235,E2 10743.235} C_VEL
LIN {X 0,Y 208.37,Z 469.791,A -85,B 0,C 180,E1 10738.991,E2 10738.991} C_VEL
LIN {X 0,Y 204.398,Z 478.178,A -85,B 0,C 180,E1 10734.264,E2 10734.264} C_VEL
LIN {X 0,Y 201.793,Z 485.071,A -85,B 0,C 180,E1 10729.09,E2 10729.09} C_VEL
LIN {X 0,Y 200.812,Z 490.059,A -85,B 0,C 180,E1 10723.829,E2 10723.829} C_VEL
LIN {X 0,Y 201.211,Z 493.253,A -85,B 0,C 180,E1 10718.558,E2 10718.558} C_VEL
LIN {X 0,Y 202.404,Z 494.619,A -85,B 0,C 180,E1 10713.753,E2 10713.753} C_VEL
LIN {X 0,Y 203.105,Z 494.514,A -85,B 0,C 180,E1 10710.284,E2 10710.284} C_VEL
LIN {X 0,Y 202.695,Z 493.776,A -85,B 0,C 180,E1 10706.892,E2 10706.892} C_VEL
LIN {X 0,Y 201.602,Z 492.372,A -85,B 0,C 180,E1 10702.705,E2 10702.705} C_VEL
LIN {X 0,Y 200.996,Z 489.182,A -85,B 0,C 180,E1 10698.514,E2 10698.514} C_VEL
LIN {X 0,Y 201.135,Z 484.374,A -85,B 0,C 180,E1 10694.431,E2 10694.431} C_VEL
LIN {X 0,Y 202.238,Z 477.034,A -85,B 0,C 180,E1 10690.057,E2 10690.057} C_VEL
LIN {X 0,Y 204.199,Z 467.808,A -85,B 0,C 180,E1 10686.023,E2 10686.023} C_VEL
LIN {X 0,Y 206.563,Z 457.587,A -85,B 0,C 180,E1 10682.626,E2 10682.626} C_VEL
LIN {X 0,Y 212.537,Z 436.015,A -85,B 0,C 180,E1 10676.769,E2 10676.769} C_VEL
LIN {X 0,Y 216.627,Z 421.857,A -85,B 0,C 180,E1 10673.79,E2 10673.79} C_VEL
LIN {X 0,Y 220.694,Z 406.806,A -85,B 0,C 180,E1 10671.306,E2 10671.306} C_VEL
LIN {X 0,Y 224.499,Z 390.92,A -85,B 0,C 180,E1 10669.275,E2 10669.275} C_VEL
LIN {X 0,Y 227.903,Z 374.21,A -85,B 0,C 180,E1 10667.671,E2 10667.671} C_VEL
LIN {X 0,Y 230.649,Z 356.514,A -85,B 0,C 180,E1 10666.455,E2 10666.455} C_VEL
LIN {X 0,Y 232.346,Z 338.442,A -85,B 0,C 180,E1 10665.634,E2 10665.634} C_VEL
LIN {X 0,Y 240.765,Z 183.778,A -85,B 0,C 180,E1 10661.145,E2 10661.145} C_VEL
LIN {X 0,Y 240.573,Z 174.869,A -85,B 0,C 180,E1 10660.758,E2 10660.758} C_VEL
LIN {X 0,Y 233.14,Z 160.106,A -85,B 0,C 180,E1 10658.766,E2 10658.766} C_VEL
LIN {X 0,Y 226.385,Z 143.328,A -85,B 0,C 180,E1 10654.77,E2 10654.77} C_VEL
LIN {X 0,Y 222.995,Z 135.364,A -85,B 0,C 180,E1 10652.551,E2 10652.551} C_VEL
LIN {X 0,Y 219.014,Z 123.503,A -85,B 0,C 180,E1 10648.263,E2 10648.263} C_VEL
LIN {X 0,Y 216.746,Z 116.269,A -85,B 0,C 180,E1 10645.185,E2 10645.185} C_VEL
LIN {X 0,Y 216.017,Z 114.425,A -85,B 0,C 180,E1 10644.181,E2 10644.181} C_VEL
LIN {X 0,Y 213.49,Z 110.807,A -85,B 0,C 180,E1 10640.994,E2 10640.994} C_VEL
LIN {X 0,Y 212.759,Z 109.302,A -85,B 0,C 180,E1 10639.777,E2 10639.777} C_VEL
LIN {X 0,Y 208.408,Z 104.05,A -85,B 0,C 180,E1 10628.791,E2 10628.791} C_VEL
LIN {X 0,Y 208.17,Z 103.85,A -85,B 0,C 180,E1 10624.131,E2 10624.131} C_VEL
LIN {X 0,Y 208.836,Z 105.828,A -85,B 0,C 180,E1 10618.902,E2 10618.902} C_VEL
LIN {X 0,Y 212.176,Z 109.443,A -85,B 0,C 180,E1 10611.872,E2 10611.872} C_VEL
LIN {X 0,Y 214.222,Z 113.364,A -85,B 0,C 180,E1 10608.422,E2 10608.422} C_VEL
LIN {X 0,Y 215.746,Z 114.933,A -85,B 0,C 180,E1 10606.601,E2 10606.601} C_VEL
LIN {X 0,Y 217.819,Z 119.003,A -85,B 0,C 180,E1 10603.739,E2 10603.739} C_VEL
LIN {X 0,Y 218.796,Z 120.255,A -85,B 0,C 180,E1 10602.72,E2 10602.72} C_VEL
LIN {X 0,Y 221.834,Z 125.891,A -85,B 0,C 180,E1 10599.416,E2 10599.416} C_VEL
LIN {X 0,Y 224.371,Z 130.723,A -85,B 0,C 180,E1 10596.911,E2 10596.911} C_VEL
LIN {X 0,Y 227.852,Z 137.673,A -85,B 0,C 180,E1 10593.691,E2 10593.691} C_VEL
LIN {X 0,Y 232.507,Z 148.648,A -85,B 0,C 180,E1 10589.506,E2 10589.506} C_VEL
LIN {X 0,Y 236.749,Z 160.251,A -85,B 0,C 180,E1 10585.826,E2 10585.826} C_VEL
LIN {X 0,Y 240.216,Z 172.654,A -85,B 0,C 180,E1 10582.425,E2 10582.425} C_VEL
LIN {X 0,Y 241.44,Z 178.968,A -85,B 0,C 180,E1 10580.935,E2 10580.935} C_VEL
LIN {X 0,Y 237.135,Z 216.32,A -85,B 0,C 180,E1 10575.661,E2 10575.661} C_VEL
LIN {X 0,Y 236.552,Z 223.113,A -85,B 0,C 180,E1 10574.768,E2 10574.768} C_VEL
LIN {X 0,Y 237.207,Z 229.84,A -85,B 0,C 180,E1 10574.353,E2 10574.353} C_VEL
LIN {X 0,Y 232.705,Z 316.76,A -85,B 0,C 180,E1 10571.847,E2 10571.847} C_VEL
LIN {X 0,Y 232.052,Z 340.016,A -85,B 0,C 180,E1 10570.952,E2 10570.952} C_VEL
LIN {X 0,Y 230.905,Z 353.93,A -85,B 0,C 180,E1 10570.028,E2 10570.028} C_VEL
LIN {X 0,Y 228.876,Z 368.037,A -85,B 0,C 180,E1 10568.657,E2 10568.657} C_VEL
LIN {X 0,Y 226.233,Z 380.963,A -85,B 0,C 180,E1 10566.943,E2 10566.943} C_VEL
LIN {X 0,Y 223.129,Z 392.938,A -85,B 0,C 180,E1 10564.84,E2 10564.84} C_VEL
LIN {X 0,Y 219.513,Z 404.328,A -85,B 0,C 180,E1 10562.2,E2 10562.2} C_VEL
LIN {X 0,Y 216.04,Z 413.621,A -85,B 0,C 180,E1 10559.376,E2 10559.376} C_VEL
LIN {X 0,Y 212.696,Z 421.564,A -85,B 0,C 180,E1 10556.221,E2 10556.221} C_VEL
LIN {X 0,Y 209.423,Z 428.495,A -85,B 0,C 180,E1 10552.452,E2 10552.452} C_VEL
LIN {X 0,Y 206.849,Z 433.336,A -85,B 0,C 180,E1 10548.602,E2 10548.602} C_VEL
LIN {X 0,Y 204.983,Z 436.415,A -85,B 0,C 180,E1 10544.691,E2 10544.691} C_VEL
LIN {X 0,Y 203.718,Z 437.915,A -85,B 0,C 180,E1 10540.46,E2 10540.46} C_VEL
LIN {X 0,Y 203.145,Z 437.514,A -85,B 0,C 180,E1 10535.93,E2 10535.93} C_VEL
LIN {X 0,Y 203.295,Z 435.286,A -85,B 0,C 180,E1 10531.689,E2 10531.689} C_VEL
LIN {X 0,Y 204.039,Z 431.544,A -85,B 0,C 180,E1 10527.751,E2 10527.751} C_VEL
LIN {X 0,Y 205.378,Z 426.001,A -85,B 0,C 180,E1 10523.85,E2 10523.85} C_VEL
LIN {X 0,Y 207.337,Z 418.337,A -85,B 0,C 180,E1 10520.001,E2 10520.001} C_VEL
LIN {X 0,Y 209.513,Z 409.706,A -85,B 0,C 180,E1 10516.756,E2 10516.756} C_VEL
LIN {X 0,Y 211.892,Z 399.655,A -85,B 0,C 180,E1 10513.833,E2 10513.833} C_VEL
LIN {X 0,Y 212.533,Z 397.448,A -85,B 0,C 180,E1 10513.181,E2 10513.181} C_VEL
LIN {X 0,Y 212.884,Z 397.408,A -85,B 0,C 180,E1 10512.928,E2 10512.928} C_VEL
LIN {X 0,Y 209.586,Z 409.18,A -85,B 0,C 180,E1 10509.238,E2 10509.238} C_VEL
LIN {X 0,Y 207.003,Z 418.622,A -85,B 0,C 180,E1 10505.454,E2 10505.454} C_VEL
LIN {X 0,Y 205.013,Z 426.28,A -85,B 0,C 180,E1 10501.388,E2 10501.388} C_VEL
LIN {X 0,Y 203.727,Z 432.316,A -85,B 0,C 180,E1 10497.061,E2 10497.061} C_VEL
LIN {X 0,Y 203.191,Z 436.368,A -85,B 0,C 180,E1 10492.751,E2 10492.751} C_VEL
LIN {X 0,Y 203.435,Z 438.925,A -85,B 0,C 180,E1 10488.053,E2 10488.053} C_VEL
LIN {X 0,Y 204.496,Z 439.543,A -85,B 0,C 180,E1 10483.584,E2 10483.584} C_VEL
LIN {X 0,Y 206.63,Z 438.317,A -85,B 0,C 180,E1 10478.823,E2 10478.823} C_VEL
LIN {X 0,Y 209.514,Z 435.433,A -85,B 0,C 180,E1 10474.605,E2 10474.605} C_VEL
LIN {X 0,Y 213.443,Z 430.58,A -85,B 0,C 180,E1 10470.393,E2 10470.393} C_VEL
LIN {X 0,Y 218.032,Z 424.226,A -85,B 0,C 180,E1 10466.587,E2 10466.587} C_VEL
LIN {X 0,Y 223.3,Z 415.933,A -85,B 0,C 180,E1 10463.017,E2 10463.017} C_VEL
LIN {X 0,Y 228.987,Z 405.935,A -85,B 0,C 180,E1 10459.782,E2 10459.782} C_VEL
LIN {X 0,Y 234.7,Z 394.442,A -85,B 0,C 180,E1 10456.967,E2 10456.967} C_VEL
LIN {X 0,Y 240.113,Z 381.994,A -85,B 0,C 180,E1 10454.605,E2 10454.605} C_VEL
LIN {X 0,Y 245.086,Z 368.462,A -85,B 0,C 180,E1 10452.619,E2 10452.619} C_VEL
LIN {X 0,Y 249.521,Z 353.709,A -85,B 0,C 180,E1 10450.961,E2 10450.961} C_VEL
LIN {X 0,Y 253.191,Z 338.231,A -85,B 0,C 180,E1 10449.651,E2 10449.651} C_VEL
LIN {X 0,Y 256.061,Z 321.182,A -85,B 0,C 180,E1 10448.626,E2 10448.626} C_VEL
LIN {X 0,Y 258.798,Z 295.92,A -85,B 0,C 180,E1 10447.671,E2 10447.671} C_VEL
LIN {X 0,Y 265.156,Z 235.817,A -85,B 0,C 180,E1 10445.735,E2 10445.735} C_VEL
LIN {X 0,Y 264.133,Z 212.438,A -85,B 0,C 180,E1 10443.554,E2 10443.554} C_VEL
LIN {X 0,Y 263.767,Z 207.817,A -85,B 0,C 180,E1 10443.015,E2 10443.015} C_VEL
LIN {X 0,Y 261.424,Z 202.188,A -85,B 0,C 180,E1 10441.412,E2 10441.412} C_VEL
LIN {X 0,Y 259.19,Z 199.131,A -85,B 0,C 180,E1 10439.917,E2 10439.917} C_VEL
LIN {X 0,Y 255.495,Z 196.786,A -85,B 0,C 180,E1 10437.344,E2 10437.344} C_VEL
LIN {X 0,Y 252.386,Z 194.442,A -85,B 0,C 180,E1 10434.537,E2 10434.537} C_VEL
LIN {X 0,Y 251.901,Z 193.581,A -85,B 0,C 180,E1 10433.935,E2 10433.935} C_VEL
LIN {X 0,Y 250.666,Z 190.891,A -85,B 0,C 180,E1 10432.091,E2 10432.091} C_VEL
LIN {X 0,Y 249.082,Z 187.771,A -85,B 0,C 180,E1 10428.774,E2 10428.774} C_VEL
LIN {X 0,Y 248.607,Z 186.395,A -85,B 0,C 180,E1 10426.73,E2 10426.73} C_VEL
LIN {X 0,Y 248.625,Z 185.738,A -85,B 0,C 180,E1 10422.687,E2 10422.687} C_VEL
LIN {X 0,Y 249.972,Z 187.164,A -85,B 0,C 180,E1 10418.747,E2 10418.747} C_VEL
LIN {X 0,Y 251.608,Z 189.004,A -85,B 0,C 180,E1 10416.213,E2 10416.213} C_VEL
LIN {X 0,Y 254.067,Z 192.801,A -85,B 0,C 180,E1 10413.344,E2 10413.344} C_VEL
LIN {X 0,Y 256.531,Z 196.632,A -85,B 0,C 180,E1 10411.099,E2 10411.099} C_VEL
LIN {X 0,Y 260,Z 202.662,A -85,B 0,C 180,E1 10408.466,E2 10408.466} C_VEL
LIN {X 0,Y 264.015,Z 210.448,A -85,B 0,C 180,E1 10405.91,E2 10405.91} C_VEL
LIN {X 0,Y 264.482,Z 211.92,A -85,B 0,C 180,E1 10405.592,E2 10405.592} C_VEL
LIN {X 0,Y 252.728,Z 338.047,A -85,B 0,C 180,E1 10402.108,E2 10402.108} C_VEL
LIN {X 0,Y 249.434,Z 357.096,A -85,B 0,C 180,E1 10401.277,E2 10401.277} C_VEL
LIN {X 0,Y 245.22,Z 373.907,A -85,B 0,C 180,E1 10400.229,E2 10400.229} C_VEL
LIN {X 0,Y 239.902,Z 390.372,A -85,B 0,C 180,E1 10398.814,E2 10398.814} C_VEL
LIN {X 0,Y 233.824,Z 406.043,A -85,B 0,C 180,E1 10396.99,E2 10396.99} C_VEL
LIN {X 0,Y 226.998,Z 421.297,A -85,B 0,C 180,E1 10394.634,E2 10394.634} C_VEL
LIN {X 0,Y 220.096,Z 435.176,A -85,B 0,C 180,E1 10391.839,E2 10391.839} C_VEL
LIN {X 0,Y 213.36,Z 447.658,A -85,B 0,C 180,E1 10388.557,E2 10388.557} C_VEL
LIN {X 0,Y 207.042,Z 458.806,A -85,B 0,C 180,E1 10384.742,E2 10384.742} C_VEL
LIN {X 0,Y 201.225,Z 469.154,A -85,B 0,C 180,E1 10380.125,E2 10380.125} C_VEL
LIN {X 0,Y 196.92,Z 477.412,A -85,B 0,C 180,E1 10375.248,E2 10375.248} C_VEL
LIN {X 0,Y 194.038,Z 484.181,A -85,B 0,C 180,E1 10369.884,E2 10369.884} C_VEL
LIN {X 0,Y 192.851,Z 489.199,A -85,B 0,C 180,E1 10364.184,E2 10364.184} C_VEL
LIN {X 0,Y 193.236,Z 492.262,A -85,B 0,C 180,E1 10358.632,E2 10358.632} C_VEL
LIN {X 0,Y 194.522,Z 493.468,A -85,B 0,C 180,E1 10353.538,E2 10353.538} C_VEL
LIN {X 0,Y 195.214,Z 493.266,A -85,B 0,C 180,E1 10350.002,E2 10350.002} C_VEL
LIN {X 0,Y 194.786,Z 492.715,A -85,B 0,C 180,E1 10347.06,E2 10347.06} C_VEL
LIN {X 0,Y 193.671,Z 491.528,A -85,B 0,C 180,E1 10342.885,E2 10342.885} C_VEL
LIN {X 0,Y 193.002,Z 488.444,A -85,B 0,C 180,E1 10338.346,E2 10338.346} C_VEL
LIN {X 0,Y 193.225,Z 483.385,A -85,B 0,C 180,E1 10333.777,E2 10333.777} C_VEL
LIN {X 0,Y 194.465,Z 476.321,A -85,B 0,C 180,E1 10329.352,E2 10329.352} C_VEL
LIN {X 0,Y 196.326,Z 468.394,A -85,B 0,C 180,E1 10325.64,E2 10325.64} C_VEL
LIN {X 0,Y 198.816,Z 458.691,A -85,B 0,C 180,E1 10322.118,E2 10322.118} C_VEL
LIN {X 0,Y 201.67,Z 447.369,A -85,B 0,C 180,E1 10318.964,E2 10318.964} C_VEL
LIN {X 0,Y 203.98,Z 438.789,A -85,B 0,C 180,E1 10316.873,E2 10316.873} C_VEL
LIN {X 0,Y 208.245,Z 424.798,A -85,B 0,C 180,E1 10313.636,E2 10313.636} C_VEL
LIN {X 0,Y 212.602,Z 409.644,A -85,B 0,C 180,E1 10310.894,E2 10310.894} C_VEL
LIN {X 0,Y 216.635,Z 393.852,A -85,B 0,C 180,E1 10308.703,E2 10308.703} C_VEL
LIN {X 0,Y 220.308,Z 376.975,A -85,B 0,C 180,E1 10306.944,E2 10306.944} C_VEL
LIN {X 0,Y 223.387,Z 358.953,A -85,B 0,C 180,E1 10305.594,E2 10305.594} C_VEL
LIN {X 0,Y 225.371,Z 340.754,A -85,B 0,C 180,E1 10304.669,E2 10304.669} C_VEL
LIN {X 0,Y 234.312,Z 184.224,A -85,B 0,C 180,E1 10300.006,E2 10300.006} C_VEL
LIN {X 0,Y 234.148,Z 177.719,A -85,B 0,C 180,E1 10299.712,E2 10299.712} C_VEL
LIN {X 0,Y 225.284,Z 160.1,A -85,B 0,C 180,E1 10297.127,E2 10297.127} C_VEL
LIN {X 0,Y 219.775,Z 143.436,A -85,B 0,C 180,E1 10292.314,E2 10292.314} C_VEL
LIN {X 0,Y 215.541,Z 130.091,A -85,B 0,C 180,E1 10287.488,E2 10287.488} C_VEL
LIN {X 0,Y 213.294,Z 122.425,A -85,B 0,C 180,E1 10284.142,E2 10284.142} C_VEL
LIN {X 0,Y 212.45,Z 121.116,A -85,B 0,C 180,E1 10283.139,E2 10283.139} C_VEL
LIN {X 0,Y 210.032,Z 116.768,A -85,B 0,C 180,E1 10279.465,E2 10279.465} C_VEL
LIN {X 0,Y 205.769,Z 111.533,A -85,B 0,C 180,E1 10268.382,E2 10268.382} C_VEL
LIN {X 0,Y 205.602,Z 111.519,A -85,B 0,C 180,E1 10263.624,E2 10263.624} C_VEL
LIN {X 0,Y 208.907,Z 116.348,A -85,B 0,C 180,E1 10252.575,E2 10252.575} C_VEL
LIN {X 0,Y 210.782,Z 120.47,A -85,B 0,C 180,E1 10248.785,E2 10248.785} C_VEL
LIN {X 0,Y 212.212,Z 122.155,A -85,B 0,C 180,E1 10246.928,E2 10246.928} C_VEL
LIN {X 0,Y 214.537,Z 126.391,A -85,B 0,C 180,E1 10243.761,E2 10243.761} C_VEL
LIN {X 0,Y 217.6,Z 132.123,A -85,B 0,C 180,E1 10240.121,E2 10240.121} C_VEL
LIN {X 0,Y 220.465,Z 138.015,A -85,B 0,C 180,E1 10237.014,E2 10237.014} C_VEL
LIN {X 0,Y 223.6,Z 144.588,A -85,B 0,C 180,E1 10233.994,E2 10233.994} C_VEL
LIN {X 0,Y 227.793,Z 154.921,A -85,B 0,C 180,E1 10229.974,E2 10229.974} C_VEL
LIN {X 0,Y 231.823,Z 166.665,A -85,B 0,C 180,E1 10226.193,E2 10226.193} C_VEL
LIN {X 0,Y 235.025,Z 178.882,A -85,B 0,C 180,E1 10222.835,E2 10222.835} C_VEL
LIN {X 0,Y 235.609,Z 182.269,A -85,B 0,C 180,E1 10222.023,E2 10222.023} C_VEL
LIN {X 0,Y 231.102,Z 218.632,A -85,B 0,C 180,E1 10216.818,E2 10216.818} C_VEL
LIN {X 0,Y 230.607,Z 224.184,A -85,B 0,C 180,E1 10216.084,E2 10216.084} C_VEL
LIN {X 0,Y 231.243,Z 231.085,A -85,B 0,C 180,E1 10215.643,E2 10215.643} C_VEL
LIN {X 0,Y 226.553,Z 317.127,A -85,B 0,C 180,E1 10213.121,E2 10213.121} C_VEL
LIN {X 0,Y 225.812,Z 341.07,A -85,B 0,C 180,E1 10212.18,E2 10212.18} C_VEL
LIN {X 0,Y 224.519,Z 355.68,A -85,B 0,C 180,E1 10211.182,E2 10211.182} C_VEL
LIN {X 0,Y 222.243,Z 370.288,A -85,B 0,C 180,E1 10209.703,E2 10209.703} C_VEL
LIN {X 0,Y 219.464,Z 382.894,A -85,B 0,C 180,E1 10207.952,E2 10207.952} C_VEL
LIN {X 0,Y 216.208,Z 394.679,A -85,B 0,C 180,E1 10205.8,E2 10205.8} C_VEL
LIN {X 0,Y 212.399,Z 406.001,A -85,B 0,C 180,E1 10203.077,E2 10203.077} C_VEL
LIN {X 0,Y 208.462,Z 415.862,A -85,B 0,C 180,E1 10199.919,E2 10199.919} C_VEL
LIN {X 0,Y 204.987,Z 423.512,A -85,B 0,C 180,E1 10196.66,E2 10196.66} C_VEL
LIN {X 0,Y 201.818,Z 429.817,A -85,B 0,C 180,E1 10193.038,E2 10193.038} C_VEL
LIN {X 0,Y 198.946,Z 434.874,A -85,B 0,C 180,E1 10188.76,E2 10188.76} C_VEL
LIN {X 0,Y 196.914,Z 437.888,A -85,B 0,C 180,E1 10184.404,E2 10184.404} C_VEL
LIN {X 0,Y 195.688,Z 439.06,A -85,B 0,C 180,E1 10180.002,E2 10180.002} C_VEL
LIN {X 0,Y 195.204,Z 438.465,A -85,B 0,C 180,E1 10175.583,E2 10175.583} C_VEL
LIN {X 0,Y 195.427,Z 436.067,A -85,B 0,C 180,E1 10171.17,E2 10171.17} C_VEL
LIN {X 0,Y 196.359,Z 431.765,A -85,B 0,C 180,E1 10166.787,E2 10166.787} C_VEL
LIN {X 0,Y 197.757,Z 426.346,A -85,B 0,C 180,E1 10163.028,E2 10163.028} C_VEL
LIN {X 0,Y 199.727,Z 419.096,A -85,B 0,C 180,E1 10159.324,E2 10159.324} C_VEL
LIN {X 0,Y 202.042,Z 410.354,A -85,B 0,C 180,E1 10155.965,E2 10155.965} C_VEL
LIN {X 0,Y 204.493,Z 401.085,A -85,B 0,C 180,E1 10153.085,E2 10153.085} C_VEL
LIN {X 0,Y 204.533,Z 401.185,A -85,B 0,C 180,E1 10152.795,E2 10152.795} C_VEL
LIN {X 0,Y 201.308,Z 412.198,A -85,B 0,C 180,E1 10149.031,E2 10149.031} C_VEL
LIN {X 0,Y 198.665,Z 421.437,A -85,B 0,C 180,E1 10144.949,E2 10144.949} C_VEL
LIN {X 0,Y 196.81,Z 428.601,A -85,B 0,C 180,E1 10140.808,E2 10140.808} C_VEL
LIN {X 0,Y 195.641,Z 434.119,A -85,B 0,C 180,E1 10136.414,E2 10136.414} C_VEL
LIN {X 0,Y 195.236,Z 438.199,A -85,B 0,C 180,E1 10131.589,E2 10131.589} C_VEL
LIN {X 0,Y 195.709,Z 440.308,A -85,B 0,C 180,E1 10126.794,E2 10126.794} C_VEL
LIN {X 0,Y 197.115,Z 440.645,A -85,B 0,C 180,E1 10122.035,E2 10122.035} C_VEL
LIN {X 0,Y 199.54,Z 439.155,A -85,B 0,C 180,E1 10117.324,E2 10117.324} C_VEL
LIN {X 0,Y 203.106,Z 435.71,A -85,B 0,C 180,E1 10112.666,E2 10112.666} C_VEL
LIN {X 0,Y 207.414,Z 430.718,A -85,B 0,C 180,E1 10108.506,E2 10108.506} C_VEL
LIN {X 0,Y 212.398,Z 424.051,A -85,B 0,C 180,E1 10104.693,E2 10104.693} C_VEL
LIN {X 0,Y 218.405,Z 415.083,A -85,B 0,C 180,E1 10100.944,E2 10100.944} C_VEL
LIN {X 0,Y 224.231,Z 405.164,A -85,B 0,C 180,E1 10097.861,E2 10097.861} C_VEL
LIN {X 0,Y 230.223,Z 393.59,A -85,B 0,C 180,E1 10095.105,E2 10095.105} C_VEL
LIN {X 0,Y 235.829,Z 380.995,A -85,B 0,C 180,E1 10092.797,E2 10092.797} C_VEL
LIN {X 0,Y 241.489,Z 365.836,A -85,B 0,C 180,E1 10090.672,E2 10090.672} C_VEL
LIN {X 0,Y 246.049,Z 350.679,A -85,B 0,C 180,E1 10089.075,E2 10089.075} C_VEL
LIN {X 0,Y 249.727,Z 334.656,A -85,B 0,C 180,E1 10087.824,E2 10087.824} C_VEL
LIN {X 0,Y 252.388,Z 318.133,A -85,B 0,C 180,E1 10086.919,E2 10086.919} C_VEL
LIN {X 0,Y 260.541,Z 244.199,A -85,B 0,C 180,E1 10084.495,E2 10084.495} C_VEL
LIN {X 0,Y 261.199,Z 237.233,A -85,B 0,C 180,E1 10084.226,E2 10084.226} C_VEL
LIN {X 0,Y 260.546,Z 214.919,A -85,B 0,C 180,E1 10082.076,E2 10082.076} C_VEL
LIN {X 0,Y 260.367,Z 212.936,A -85,B 0,C 180,E1 10081.816,E2 10081.816} C_VEL
LIN {X 0,Y 257.388,Z 205.564,A -85,B 0,C 180,E1 10079.5,E2 10079.5} C_VEL
LIN {X 0,Y 254.164,Z 198.067,A -85,B 0,C 180,E1 10076.505,E2 10076.505} C_VEL
LIN {X 0,Y 251.901,Z 193.581,A -85,B 0,C 180,E1 10073.935,E2 10073.935} C_VEL
LIN {X 0,Y 250.712,Z 192.163,A -85,B 0,C 180,E1 10072.353,E2 10072.353} C_VEL
LIN {X 0,Y 249.068,Z 192.535,A -85,B 0,C 180,E1 10070.082,E2 10070.082} C_VEL
LIN {X 0,Y 247.396,Z 194.11,A -85,B 0,C 180,E1 10066.573,E2 10066.573} C_VEL
LIN {X 0,Y 247.263,Z 194.021,A -85,B 0,C 180,E1 10065.785,E2 10065.785} C_VEL
LIN {X 0,Y 247.526,Z 193.732,A -85,B 0,C 180,E1 10062.122,E2 10062.122} C_VEL
LIN {X 0,Y 249.422,Z 195.774,A -85,B 0,C 180,E1 10057.616,E2 10057.616} C_VEL
LIN {X 0,Y 251.851,Z 199.429,A -85,B 0,C 180,E1 10054.359,E2 10054.359} C_VEL
LIN {X 0,Y 254.617,Z 204.1,A -85,B 0,C 180,E1 10051.599,E2 10051.599} C_VEL
LIN {X 0,Y 257.788,Z 209.893,A -85,B 0,C 180,E1 10049.075,E2 10049.075} C_VEL
LIN {X 0,Y 260.692,Z 215.83,A -85,B 0,C 180,E1 10047.073,E2 10047.073} C_VEL
LIN {X 0,Y 248.688,Z 337.73,A -85,B 0,C 180,E1 10043.695,E2 10043.695} C_VEL
LIN {X 0,Y 245.324,Z 356.289,A -85,B 0,C 180,E1 10042.889,E2 10042.889} C_VEL
LIN {X 0,Y 240.938,Z 373.059,A -85,B 0,C 180,E1 10041.852,E2 10041.852} C_VEL
LIN {X 0,Y 235.371,Z 389.528,A -85,B 0,C 180,E1 10040.447,E2 10040.447} C_VEL
LIN {X 0,Y 228.766,Z 405.799,A -85,B 0,C 180,E1 10038.555,E2 10038.555} C_VEL
LIN {X 0,Y 221.913,Z 420.405,A -85,B 0,C 180,E1 10036.294,E2 10036.294} C_VEL
LIN {X 0,Y 214.778,Z 433.948,A -85,B 0,C 180,E1 10033.552,E2 10033.552} C_VEL
LIN {X 0,Y 207.544,Z 446.55,A -85,B 0,C 180,E1 10030.209,E2 10030.209} C_VEL
LIN {X 0,Y 200.793,Z 457.698,A -85,B 0,C 180,E1 10026.341,E2 10026.341} C_VEL
LIN {X 0,Y 194.491,Z 467.987,A -85,B 0,C 180,E1 10021.628,E2 10021.628} C_VEL
LIN {X 0,Y 189.738,Z 476.233,A -85,B 0,C 180,E1 10016.613,E2 10016.613} C_VEL
LIN {X 0,Y 186.452,Z 482.975,A -85,B 0,C 180,E1 10011.059,E2 10011.059} C_VEL
LIN {X 0,Y 184.934,Z 488.032,A -85,B 0,C 180,E1 10005.043,E2 10005.043} C_VEL
LIN {X 0,Y 185.219,Z 491.192,A -85,B 0,C 180,E1 9998.933,E2 9998.933} C_VEL
LIN {X 0,Y 186.534,Z 492.293,A -85,B 0,C 180,E1 9993.69,E2 9993.69} C_VEL
LIN {X 0,Y 187.305,Z 492.054,A -85,B 0,C 180,E1 9990.002,E2 9990.002} C_VEL
LIN {X 0,Y 186.967,Z 491.622,A -85,B 0,C 180,E1 9987.55,E2 9987.55} C_VEL
LIN {X 0,Y 185.77,Z 490.738,A -85,B 0,C 180,E1 9983.202,E2 9983.202} C_VEL
LIN {X 0,Y 185.01,Z 487.68,A -85,B 0,C 180,E1 9978.152,E2 9978.152} C_VEL
LIN {X 0,Y 185.284,Z 482.773,A -85,B 0,C 180,E1 9973.384,E2 9973.384} C_VEL
LIN {X 0,Y 186.438,Z 476.795,A -85,B 0,C 180,E1 9969.273,E2 9969.273} C_VEL
LIN {X 0,Y 188.65,Z 468.254,A -85,B 0,C 180,E1 9964.915,E2 9964.915} C_VEL
LIN {X 0,Y 191.576,Z 457.902,A -85,B 0,C 180,E1 9960.966,E2 9960.966} C_VEL
LIN {X 0,Y 194.85,Z 446.111,A -85,B 0,C 180,E1 9957.576,E2 9957.576} C_VEL
LIN {X 0,Y 197.995,Z 433.658,A -85,B 0,C 180,E1 9954.855,E2 9954.855} C_VEL
LIN {X 0,Y 203.329,Z 416.159,A -85,B 0,C 180,E1 9951.176,E2 9951.176} C_VEL
LIN {X 0,Y 207.655,Z 400.813,A -85,B 0,C 180,E1 9948.689,E2 9948.689} C_VEL
LIN {X 0,Y 211.702,Z 384.307,A -85,B 0,C 180,E1 9946.663,E2 9946.663} C_VEL
LIN {X 0,Y 215.224,Z 366.749,A -85,B 0,C 180,E1 9945.082,E2 9945.082} C_VEL
LIN {X 0,Y 217.78,Z 348.964,A -85,B 0,C 180,E1 9943.958,E2 9943.958} C_VEL
LIN {X 0,Y 219.271,Z 330.195,A -85,B 0,C 180,E1 9943.212,E2 9943.212} C_VEL
LIN {X 0,Y 227.926,Z 184.768,A -85,B 0,C 180,E1 9938.818,E2 9938.818} C_VEL
LIN {X 0,Y 227.759,Z 180.608,A -85,B 0,C 180,E1 9938.607,E2 9938.607} C_VEL
LIN {X 0,Y 221.441,Z 167.729,A -85,B 0,C 180,E1 9936.665,E2 9936.665} C_VEL
LIN {X 0,Y 217.571,Z 155.114,A -85,B 0,C 180,E1 9933.152,E2 9933.152} C_VEL
LIN {X 0,Y 213.9,Z 143.099,A -85,B 0,C 180,E1 9929.163,E2 9929.163} C_VEL
LIN {X 0,Y 211.168,Z 133.24,A -85,B 0,C 180,E1 9925.222,E2 9925.222} C_VEL
LIN {X 0,Y 209.924,Z 128.814,A -85,B 0,C 180,E1 9923.137,E2 9923.137} C_VEL
LIN {X 0,Y 207.366,Z 124.565,A -85,B 0,C 180,E1 9919.505,E2 9919.505} C_VEL
LIN {X 0,Y 203.045,Z 119.088,A -85,B 0,C 180,E1 9908.495,E2 9908.495} C_VEL
LIN {X 0,Y 202.758,Z 119.001,A -85,B 0,C 180,E1 9903.675,E2 9903.675} C_VEL
LIN {X 0,Y 205.616,Z 123.591,A -85,B 0,C 180,E1 9892.876,E2 9892.876} C_VEL
LIN {X 0,Y 207.576,Z 127.815,A -85,B 0,C 180,E1 9888.891,E2 9888.891} C_VEL
LIN {X 0,Y 208.732,Z 129.37,A -85,B 0,C 180,E1 9887.27,E2 9887.27} C_VEL
LIN {X 0,Y 211.248,Z 134.247,A -85,B 0,C 180,E1 9883.501,E2 9883.501} C_VEL
LIN {X 0,Y 213.719,Z 139.323,A -85,B 0,C 180,E1 9880.315,E2 9880.315} C_VEL
LIN {X 0,Y 217.059,Z 146.123,A -85,B 0,C 180,E1 9876.662,E2 9876.662} C_VEL
LIN {X 0,Y 221.321,Z 156.35,A -85,B 0,C 180,E1 9872.268,E2 9872.268} C_VEL
LIN {X 0,Y 225.101,Z 167.236,A -85,B 0,C 180,E1 9868.389,E2 9868.389} C_VEL
LIN {X 0,Y 228.364,Z 178.756,A -85,B 0,C 180,E1 9864.955,E2 9864.955} C_VEL
LIN {X 0,Y 229.803,Z 186.022,A -85,B 0,C 180,E1 9863.099,E2 9863.099} C_VEL
LIN {X 0,Y 224.907,Z 222.809,A -85,B 0,C 180,E1 9857.763,E2 9857.763} C_VEL
LIN {X 0,Y 224.826,Z 225.567,A -85,B 0,C 180,E1 9857.447,E2 9857.447} C_VEL
LIN {X 0,Y 225.395,Z 232.414,A -85,B 0,C 180,E1 9856.999,E2 9856.999} C_VEL
LIN {X 0,Y 220.517,Z 317.666,A -85,B 0,C 180,E1 9854.46,E2 9854.46} C_VEL
LIN {X 0,Y 219.673,Z 342.283,A -85,B 0,C 180,E1 9853.468,E2 9853.468} C_VEL
LIN {X 0,Y 218.269,Z 357.05,A -85,B 0,C 180,E1 9852.432,E2 9852.432} C_VEL
LIN {X 0,Y 215.916,Z 371.341,A -85,B 0,C 180,E1 9850.953,E2 9850.953} C_VEL
LIN {X 0,Y 212.972,Z 384.041,A -85,B 0,C 180,E1 9849.154,E2 9849.154} C_VEL
LIN {X 0,Y 209.547,Z 395.815,A -85,B 0,C 180,E1 9846.953,E2 9846.953} C_VEL
LIN {X 0,Y 205.678,Z 406.758,A -85,B 0,C 180,E1 9844.266,E2 9844.266} C_VEL
LIN {X 0,Y 201.881,Z 415.87,A -85,B 0,C 180,E1 9841.332,E2 9841.332} C_VEL
LIN {X 0,Y 198.147,Z 423.801,A -85,B 0,C 180,E1 9837.985,E2 9837.985} C_VEL
LIN {X 0,Y 194.469,Z 430.723,A -85,B 0,C 180,E1 9833.962,E2 9833.962} C_VEL
LIN {X 0,Y 191.379,Z 435.84,A -85,B 0,C 180,E1 9829.531,E2 9829.531} C_VEL
LIN {X 0,Y 189.181,Z 438.917,A -85,B 0,C 180,E1 9825.007,E2 9825.007} C_VEL
LIN {X 0,Y 187.834,Z 440.15,A -85,B 0,C 180,E1 9820.425,E2 9820.425} C_VEL
LIN {X 0,Y 187.284,Z 439.612,A -85,B 0,C 180,E1 9815.819,E2 9815.819} C_VEL
LIN {X 0,Y 187.527,Z 437.046,A -85,B 0,C 180,E1 9810.914,E2 9810.914} C_VEL
LIN {X 0,Y 188.537,Z 432.671,A -85,B 0,C 180,E1 9806.349,E2 9806.349} C_VEL
LIN {X 0,Y 190.177,Z 426.669,A -85,B 0,C 180,E1 9802.141,E2 9802.141} C_VEL
LIN {X 0,Y 192.33,Z 419.166,A -85,B 0,C 180,E1 9798.3,E2 9798.3} C_VEL
LIN {X 0,Y 194.843,Z 410.182,A -85,B 0,C 180,E1 9794.826,E2 9794.826} C_VEL
LIN {X 0,Y 196.499,Z 404.486,A -85,B 0,C 180,E1 9792.928,E2 9792.928} C_VEL
LIN {X 0,Y 195.848,Z 405.667,A -85,B 0,C 180,E1 9792.314,E2 9792.314} C_VEL
LIN {X 0,Y 192.652,Z 416.307,A -85,B 0,C 180,E1 9788.282,E2 9788.282} C_VEL
LIN {X 0,Y 190.204,Z 424.67,A -85,B 0,C 180,E1 9784.129,E2 9784.129} C_VEL
LIN {X 0,Y 188.345,Z 431.914,A -85,B 0,C 180,E1 9779.318,E2 9779.318} C_VEL
LIN {X 0,Y 187.444,Z 436.82,A -85,B 0,C 180,E1 9774.701,E2 9774.701} C_VEL
LIN {X 0,Y 187.373,Z 440.2,A -85,B 0,C 180,E1 9769.737,E2 9769.737} C_VEL
LIN {X 0,Y 188.192,Z 441.774,A -85,B 0,C 180,E1 9764.962,E2 9764.962} C_VEL
LIN {X 0,Y 190.124,Z 441.563,A -85,B 0,C 180,E1 9759.84,E2 9759.84} C_VEL
LIN {X 0,Y 193.058,Z 439.623,A -85,B 0,C 180,E1 9755.083,E2 9755.083} C_VEL
LIN {X 0,Y 197.075,Z 435.829,A -85,B 0,C 180,E1 9750.488,E2 9750.488} C_VEL
LIN {X 0,Y 202.367,Z 429.875,A -85,B 0,C 180,E1 9745.94,E2 9745.94} C_VEL
LIN {X 0,Y 208.152,Z 422.414,A -85,B 0,C 180,E1 9742.005,E2 9742.005} C_VEL
LIN {X 0,Y 214.382,Z 413.296,A -85,B 0,C 180,E1 9738.491,E2 9738.491} C_VEL
LIN {X 0,Y 220.538,Z 403.071,A -85,B 0,C 180,E1 9735.516,E2 9735.516} C_VEL
LIN {X 0,Y 226.695,Z 391.351,A -85,B 0,C 180,E1 9732.901,E2 9732.901} C_VEL
LIN {X 0,Y 232.59,Z 378.303,A -85,B 0,C 180,E1 9730.653,E2 9730.653} C_VEL
LIN {X 0,Y 237.784,Z 364.482,A -85,B 0,C 180,E1 9728.823,E2 9728.823} C_VEL
LIN {X 0,Y 242.646,Z 348.28,A -85,B 0,C 180,E1 9727.209,E2 9727.209} C_VEL
LIN {X 0,Y 246.329,Z 332.024,A -85,B 0,C 180,E1 9726.024,E2 9726.024} C_VEL
LIN {X 0,Y 248.993,Z 314.457,A -85,B 0,C 180,E1 9725.152,E2 9725.152} C_VEL
LIN {X 0,Y 257.555,Z 239.111,A -85,B 0,C 180,E1 9722.698,E2 9722.698} C_VEL
LIN {X 0,Y 257.203,Z 218.354,A -85,B 0,C 180,E1 9720.655,E2 9720.655} C_VEL
LIN {X 0,Y 254.159,Z 210.228,A -85,B 0,C 180,E1 9717.971,E2 9717.971} C_VEL
LIN {X 0,Y 251.63,Z 204.244,A -85,B 0,C 180,E1 9715.277,E2 9715.277} C_VEL
LIN {X 0,Y 249.202,Z 198.679,A -85,B 0,C 180,E1 9711.812,E2 9711.812} C_VEL
LIN {X 0,Y 247.631,Z 195.247,A -85,B 0,C 180,E1 9708.117,E2 9708.117} C_VEL
LIN {X 0,Y 247.343,Z 194.227,A -85,B 0,C 180,E1 9706.441,E2 9706.441} C_VEL
LIN {X 0,Y 247.263,Z 194.021,A -85,B 0,C 180,E1 9705.785,E2 9705.785} C_VEL
LIN {X 0,Y 247.104,Z 194.585,A -85,B 0,C 180,E1 9704.123,E2 9704.123} C_VEL
LIN {X 0,Y 246.976,Z 197.88,A -85,B 0,C 180,E1 9701.779,E2 9701.779} C_VEL
LIN {X 0,Y 247.576,Z 202.684,A -85,B 0,C 180,E1 9698.823,E2 9698.823} C_VEL
LIN {X 0,Y 248.083,Z 203.618,A -85,B 0,C 180,E1 9697.806,E2 9697.806} C_VEL
LIN {X 0,Y 250.283,Z 207.216,A -85,B 0,C 180,E1 9694.694,E2 9694.694} C_VEL
LIN {X 0,Y 252.77,Z 211.569,A -85,B 0,C 180,E1 9692.112,E2 9692.112} C_VEL
LIN {X 0,Y 255.537,Z 216.972,A -85,B 0,C 180,E1 9689.751,E2 9689.751} C_VEL
LIN {X 0,Y 257.012,Z 220.5,A -85,B 0,C 180,E1 9688.573,E2 9688.573} C_VEL
LIN {X 0,Y 244.985,Z 336.694,A -85,B 0,C 180,E1 9685.364,E2 9685.364} C_VEL
LIN {X 0,Y 241.434,Z 355.51,A -85,B 0,C 180,E1 9684.557,E2 9684.557} C_VEL
LIN {X 0,Y 236.866,Z 372.405,A -85,B 0,C 180,E1 9683.529,E2 9683.529} C_VEL
LIN {X 0,Y 231.104,Z 388.813,A -85,B 0,C 180,E1 9682.148,E2 9682.148} C_VEL
LIN {X 0,Y 224.564,Z 404.243,A -85,B 0,C 180,E1 9680.38,E2 9680.38} C_VEL
LIN {X 0,Y 217.104,Z 419.385,A -85,B 0,C 180,E1 9678.056,E2 9678.056} C_VEL
LIN {X 0,Y 209.289,Z 433.486,A -85,B 0,C 180,E1 9675.192,E2 9675.192} C_VEL
LIN {X 0,Y 201.924,Z 445.532,A -85,B 0,C 180,E1 9671.951,E2 9671.951} C_VEL
LIN {X 0,Y 194.716,Z 456.601,A -85,B 0,C 180,E1 9668.041,E2 9668.041} C_VEL
LIN {X 0,Y 187.906,Z 466.877,A -85,B 0,C 180,E1 9663.237,E2 9663.237} C_VEL
LIN {X 0,Y 182.676,Z 475.077,A -85,B 0,C 180,E1 9658.083,E2 9658.083} C_VEL
LIN {X 0,Y 178.951,Z 481.782,A -85,B 0,C 180,E1 9652.332,E2 9652.332} C_VEL
LIN {X 0,Y 177.097,Z 486.673,A -85,B 0,C 180,E1 9646.305,E2 9646.305} C_VEL
LIN {X 0,Y 177.082,Z 489.832,A -85,B 0,C 180,E1 9640.083,E2 9640.083} C_VEL
LIN {X 0,Y 178.351,Z 491.066,A -85,B 0,C 180,E1 9634.504,E2 9634.504} C_VEL
LIN {X 0,Y 179.327,Z 490.93,A -85,B 0,C 180,E1 9630.641,E2 9630.641} C_VEL
LIN {X 0,Y 179.155,Z 490.5,A -85,B 0,C 180,E1 9628.084,E2 9628.084} C_VEL
LIN {X 0,Y 177.885,Z 489.859,A -85,B 0,C 180,E1 9623.548,E2 9623.548} C_VEL
LIN {X 0,Y 177.085,Z 487.587,A -85,B 0,C 180,E1 9618.935,E2 9618.935} C_VEL
LIN {X 0,Y 177.192,Z 483.281,A -85,B 0,C 180,E1 9613.952,E2 9613.952} C_VEL
LIN {X 0,Y 178.362,Z 477.363,A -85,B 0,C 180,E1 9609.322,E2 9609.322} C_VEL
LIN {X 0,Y 180.403,Z 470.04,A -85,B 0,C 180,E1 9605.092,E2 9605.092} C_VEL
LIN {X 0,Y 183.352,Z 460.56,A -85,B 0,C 180,E1 9600.969,E2 9600.969} C_VEL
LIN {X 0,Y 186.829,Z 449.296,A -85,B 0,C 180,E1 9597.284,E2 9597.284} C_VEL
LIN {X 0,Y 190.253,Z 437.328,A -85,B 0,C 180,E1 9594.317,E2 9594.317} C_VEL
LIN {X 0,Y 193.451,Z 424.498,A -85,B 0,C 180,E1 9591.901,E2 9591.901} C_VEL
LIN {X 0,Y 199.293,Z 404.846,A -85,B 0,C 180,E1 9588.34,E2 9588.34} C_VEL
LIN {X 0,Y 203.516,Z 389.05,A -85,B 0,C 180,E1 9586.158,E2 9586.158} C_VEL
LIN {X 0,Y 207.264,Z 372.446,A -85,B 0,C 180,E1 9584.446,E2 9584.446} C_VEL
LIN {X 0,Y 210.29,Z 354.763,A -85,B 0,C 180,E1 9583.143,E2 9583.143} C_VEL
LIN {X 0,Y 212.176,Z 336.64,A -85,B 0,C 180,E1 9582.261,E2 9582.261} C_VEL
LIN {X 0,Y 221.629,Z 185.019,A -85,B 0,C 180,E1 9577.555,E2 9577.555} C_VEL
LIN {X 0,Y 221.338,Z 183.192,A -85,B 0,C 180,E1 9577.414,E2 9577.414} C_VEL
LIN {X 0,Y 217.569,Z 175.23,A -85,B 0,C 180,E1 9576.154,E2 9576.154} C_VEL
LIN {X 0,Y 214.949,Z 165.616,A -85,B 0,C 180,E1 9573.57,E2 9573.57} C_VEL
LIN {X 0,Y 211.006,Z 152.041,A -85,B 0,C 180,E1 9569.213,E2 9569.213} C_VEL
LIN {X 0,Y 207.909,Z 140.236,A -85,B 0,C 180,E1 9564.581,E2 9564.581} C_VEL
LIN {X 0,Y 206.729,Z 135.851,A -85,B 0,C 180,E1 9562.463,E2 9562.463} C_VEL
LIN {X 0,Y 204.259,Z 131.532,A -85,B 0,C 180,E1 9558.552,E2 9558.552} C_VEL
LIN {X 0,Y 200.389,Z 126.565,A -85,B 0,C 180,E1 9548.03,E2 9548.03} C_VEL
LIN {X 0,Y 200.105,Z 126.556,A -85,B 0,C 180,E1 9543.724,E2 9543.724} C_VEL
LIN {X 0,Y 202.582,Z 131,A -85,B 0,C 180,E1 9533.197,E2 9533.197} C_VEL
LIN {X 0,Y 204.224,Z 134.954,A -85,B 0,C 180,E1 9529.277,E2 9529.277} C_VEL
LIN {X 0,Y 205.129,Z 136.141,A -85,B 0,C 180,E1 9527.901,E2 9527.901} C_VEL
LIN {X 0,Y 207.705,Z 141.501,A -85,B 0,C 180,E1 9523.787,E2 9523.787} C_VEL
LIN {X 0,Y 209.889,Z 146.133,A -85,B 0,C 180,E1 9520.81,E2 9520.81} C_VEL
LIN {X 0,Y 213.08,Z 153.043,A -85,B 0,C 180,E1 9517.078,E2 9517.078} C_VEL
LIN {X 0,Y 216.826,Z 162.65,A -85,B 0,C 180,E1 9512.836,E2 9512.836} C_VEL
LIN {X 0,Y 220.4,Z 173.621,A -85,B 0,C 180,E1 9508.857,E2 9508.857} C_VEL
LIN {X 0,Y 223.383,Z 185.26,A -85,B 0,C 180,E1 9505.357,E2 9505.357} C_VEL
LIN {X 0,Y 224.131,Z 189.458,A -85,B 0,C 180,E1 9504.278,E2 9504.278} C_VEL
LIN {X 0,Y 219.038,Z 225.674,A -85,B 0,C 180,E1 9498.979,E2 9498.979} C_VEL
LIN {X 0,Y 219.694,Z 233.531,A -85,B 0,C 180,E1 9498.433,E2 9498.433} C_VEL
LIN {X 0,Y 214.614,Z 318.088,A -85,B 0,C 180,E1 9495.878,E2 9495.878} C_VEL
LIN {X 0,Y 213.674,Z 343.222,A -85,B 0,C 180,E1 9494.847,E2 9494.847} C_VEL
LIN {X 0,Y 212.24,Z 357.633,A -85,B 0,C 180,E1 9493.826,E2 9493.826} C_VEL
LIN {X 0,Y 209.793,Z 371.926,A -85,B 0,C 180,E1 9492.335,E2 9492.335} C_VEL
LIN {X 0,Y 206.821,Z 384.328,A -85,B 0,C 180,E1 9490.573,E2 9490.573} C_VEL
LIN {X 0,Y 203.186,Z 396.355,A -85,B 0,C 180,E1 9488.315,E2 9488.315} C_VEL
LIN {X 0,Y 198.777,Z 408.211,A -85,B 0,C 180,E1 9485.339,E2 9485.339} C_VEL
LIN {X 0,Y 194.376,Z 418.112,A -85,B 0,C 180,E1 9481.99,E2 9481.99} C_VEL
LIN {X 0,Y 190.492,Z 425.749,A -85,B 0,C 180,E1 9478.528,E2 9478.528} C_VEL
LIN {X 0,Y 186.794,Z 432.249,A -85,B 0,C 180,E1 9474.498,E2 9474.498} C_VEL
LIN {X 0,Y 183.666,Z 437.092,A -85,B 0,C 180,E1 9470.055,E2 9470.055} C_VEL
LIN {X 0,Y 181.261,Z 440.194,A -85,B 0,C 180,E1 9465.13,E2 9465.13} C_VEL
LIN {X 0,Y 179.86,Z 441.27,A -85,B 0,C 180,E1 9460.244,E2 9460.244} C_VEL
LIN {X 0,Y 179.34,Z 440.529,A -85,B 0,C 180,E1 9455.436,E2 9455.436} C_VEL
LIN {X 0,Y 179.63,Z 438.012,A -85,B 0,C 180,E1 9450.635,E2 9450.635} C_VEL
LIN {X 0,Y 180.726,Z 433.576,A -85,B 0,C 180,E1 9445.873,E2 9445.873} C_VEL
LIN {X 0,Y 182.49,Z 427.489,A -85,B 0,C 180,E1 9441.491,E2 9441.491} C_VEL
LIN {X 0,Y 184.793,Z 419.889,A -85,B 0,C 180,E1 9437.499,E2 9437.499} C_VEL
LIN {X 0,Y 187.473,Z 410.802,A -85,B 0,C 180,E1 9433.897,E2 9433.897} C_VEL
LIN {X 0,Y 188.211,Z 407.948,A -85,B 0,C 180,E1 9432.85,E2 9432.85} C_VEL
LIN {X 0,Y 187.63,Z 408.622,A -85,B 0,C 180,E1 9432.315,E2 9432.315} C_VEL
LIN {X 0,Y 184.603,Z 418.217,A -85,B 0,C 180,E1 9428.387,E2 9428.387} C_VEL
LIN {X 0,Y 182.07,Z 426.569,A -85,B 0,C 180,E1 9423.937,E2 9423.937} C_VEL
LIN {X 0,Y 180.346,Z 433.225,A -85,B 0,C 180,E1 9419.244,E2 9419.244} C_VEL
LIN {X 0,Y 179.444,Z 438.253,A -85,B 0,C 180,E1 9414.191,E2 9414.191} C_VEL
LIN {X 0,Y 179.512,Z 441.587,A -85,B 0,C 180,E1 9408.908,E2 9408.908} C_VEL
LIN {X 0,Y 180.567,Z 442.995,A -85,B 0,C 180,E1 9403.803,E2 9403.803} C_VEL
LIN {X 0,Y 182.808,Z 442.658,A -85,B 0,C 180,E1 9398.541,E2 9398.541} C_VEL
LIN {X 0,Y 186.141,Z 440.555,A -85,B 0,C 180,E1 9393.592,E2 9393.592} C_VEL
LIN {X 0,Y 190.785,Z 436.426,A -85,B 0,C 180,E1 9388.688,E2 9388.688} C_VEL
LIN {X 0,Y 196.322,Z 430.62,A -85,B 0,C 180,E1 9384.264,E2 9384.264} C_VEL
LIN {X 0,Y 202.651,Z 422.857,A -85,B 0,C 180,E1 9380.205,E2 9380.205} C_VEL
LIN {X 0,Y 209.359,Z 413.606,A -85,B 0,C 180,E1 9376.652,E2 9376.652} C_VEL
LIN {X 0,Y 216.042,Z 402.978,A -85,B 0,C 180,E1 9373.611,E2 9373.611} C_VEL
LIN {X 0,Y 222.963,Z 390.253,A -85,B 0,C 180,E1 9370.856,E2 9370.856} C_VEL
LIN {X 0,Y 229.142,Z 376.788,A -85,B 0,C 180,E1 9368.646,E2 9368.646} C_VEL
LIN {X 0,Y 234.96,Z 361.454,A -85,B 0,C 180,E1 9366.733,E2 9366.733} C_VEL
LIN {X 0,Y 239.448,Z 346.507,A -85,B 0,C 180,E1 9365.337,E2 9365.337} C_VEL
LIN {X 0,Y 243.231,Z 329.398,A -85,B 0,C 180,E1 9364.177,E2 9364.177} C_VEL
LIN {X 0,Y 245.697,Z 312.426,A -85,B 0,C 180,E1 9363.402,E2 9363.402} C_VEL
LIN {X 0,Y 254.133,Z 240.726,A -85,B 0,C 180,E1 9361.099,E2 9361.099} C_VEL
LIN {X 0,Y 254.111,Z 223.413,A -85,B 0,C 180,E1 9359.352,E2 9359.352} C_VEL
LIN {X 0,Y 251.57,Z 216.249,A -85,B 0,C 180,E1 9356.811,E2 9356.811} C_VEL
LIN {X 0,Y 249.693,Z 211.442,A -85,B 0,C 180,E1 9354.601,E2 9354.601} C_VEL
LIN {X 0,Y 247.613,Z 206.207,A -85,B 0,C 180,E1 9351.291,E2 9351.291} C_VEL
LIN {X 0,Y 246.217,Z 202.383,A -85,B 0,C 180,E1 9347.065,E2 9347.065} C_VEL
LIN {X 0,Y 246.162,Z 201.545,A -85,B 0,C 180,E1 9342.996,E2 9342.996} C_VEL
LIN {X 0,Y 247.252,Z 202.717,A -85,B 0,C 180,E1 9339.402,E2 9339.402} C_VEL
LIN {X 0,Y 248.083,Z 203.618,A -85,B 0,C 180,E1 9337.806,E2 9337.806} C_VEL
LIN {X 0,Y 248.971,Z 205.539,A -85,B 0,C 180,E1 9336.361,E2 9336.361} C_VEL
LIN {X 0,Y 249.927,Z 210.198,A -85,B 0,C 180,E1 9334.626,E2 9334.626} C_VEL
LIN {X 0,Y 252.28,Z 221.516,A -85,B 0,C 180,E1 9331.373,E2 9331.373} C_VEL
LIN {X 0,Y 252.746,Z 222.711,A -85,B 0,C 180,E1 9330.941,E2 9330.941} C_VEL
LIN {X 0,Y 253.661,Z 225.042,A -85,B 0,C 180,E1 9330.134,E2 9330.134} C_VEL
LIN {X 0,Y 241.518,Z 336.25,A -85,B 0,C 180,E1 9327.075,E2 9327.075} C_VEL
LIN {X 0,Y 237.85,Z 354.901,A -85,B 0,C 180,E1 9326.287,E2 9326.287} C_VEL
LIN {X 0,Y 233.015,Z 371.978,A -85,B 0,C 180,E1 9325.259,E2 9325.259} C_VEL
LIN {X 0,Y 227.054,Z 388.156,A -85,B 0,C 180,E1 9323.909,E2 9323.909} C_VEL
LIN {X 0,Y 219.915,Z 404.222,A -85,B 0,C 180,E1 9322.078,E2 9322.078} C_VEL
LIN {X 0,Y 212.292,Z 418.965,A -85,B 0,C 180,E1 9319.816,E2 9319.816} C_VEL
LIN {X 0,Y 204.591,Z 432.097,A -85,B 0,C 180,E1 9317.146,E2 9317.146} C_VEL
LIN {X 0,Y 196.173,Z 445.025,A -85,B 0,C 180,E1 9313.636,E2 9313.636} C_VEL
LIN {X 0,Y 188.357,Z 456.251,A -85,B 0,C 180,E1 9309.57,E2 9309.57} C_VEL
LIN {X 0,Y 181.488,Z 465.788,A -85,B 0,C 180,E1 9304.959,E2 9304.959} C_VEL
LIN {X 0,Y 175.747,Z 473.956,A -85,B 0,C 180,E1 9299.669,E2 9299.669} C_VEL
LIN {X 0,Y 171.542,Z 480.607,A -85,B 0,C 180,E1 9293.717,E2 9293.717} C_VEL
LIN {X 0,Y 169.248,Z 485.621,A -85,B 0,C 180,E1 9287.183,E2 9287.183} C_VEL
LIN {X 0,Y 169.067,Z 488.738,A -85,B 0,C 180,E1 9280.566,E2 9280.566} C_VEL
LIN {X 0,Y 170.336,Z 489.884,A -85,B 0,C 180,E1 9274.716,E2 9274.716} C_VEL
LIN {X 0,Y 171.412,Z 489.685,A -85,B 0,C 180,E1 9270.671,E2 9270.671} C_VEL
LIN {X 0,Y 171.269,Z 489.359,A -85,B 0,C 180,E1 9268.33,E2 9268.33} C_VEL
LIN {X 0,Y 169.973,Z 488.926,A -85,B 0,C 180,E1 9263.787,E2 9263.787} C_VEL
LIN {X 0,Y 169.068,Z 486.536,A -85,B 0,C 180,E1 9258.403,E2 9258.403} C_VEL
LIN {X 0,Y 169.364,Z 481.922,A -85,B 0,C 180,E1 9252.835,E2 9252.835} C_VEL
LIN {X 0,Y 170.971,Z 475.428,A -85,B 0,C 180,E1 9247.662,E2 9247.662} C_VEL
LIN {X 0,Y 173.393,Z 467.829,A -85,B 0,C 180,E1 9243.274,E2 9243.274} C_VEL
LIN {X 0,Y 176.478,Z 458.904,A -85,B 0,C 180,E1 9239.346,E2 9239.346} C_VEL
LIN {X 0,Y 180.335,Z 447.527,A -85,B 0,C 180,E1 9235.564,E2 9235.564} C_VEL
LIN {X 0,Y 184.328,Z 434.604,A -85,B 0,C 180,E1 9232.368,E2 9232.368} C_VEL
LIN {X 0,Y 187.811,Z 421.209,A -85,B 0,C 180,E1 9229.9,E2 9229.9} C_VEL
LIN {X 0,Y 190.28,Z 410.7,A -85,B 0,C 180,E1 9228.343,E2 9228.343} C_VEL
LIN {X 0,Y 195.006,Z 394.498,A -85,B 0,C 180,E1 9225.792,E2 9225.792} C_VEL
LIN {X 0,Y 199.165,Z 377.868,A -85,B 0,C 180,E1 9223.825,E2 9223.825} C_VEL
LIN {X 0,Y 202.622,Z 360.374,A -85,B 0,C 180,E1 9222.348,E2 9222.348} C_VEL
LIN {X 0,Y 205.018,Z 342.111,A -85,B 0,C 180,E1 9221.285,E2 9221.285} C_VEL
LIN {X 0,Y 207.145,Z 310.805,A -85,B 0,C 180,E1 9220.206,E2 9220.206} C_VEL
LIN {X 0,Y 215.364,Z 186.691,A -85,B 0,C 180,E1 9216.294,E2 9216.294} C_VEL
LIN {X 0,Y 213.661,Z 182.714,A -85,B 0,C 180,E1 9215.593,E2 9215.593} C_VEL
LIN {X 0,Y 211.343,Z 173.172,A -85,B 0,C 180,E1 9213.081,E2 9213.081} C_VEL
LIN {X 0,Y 207.415,Z 158.475,A -85,B 0,C 180,E1 9208.347,E2 9208.347} C_VEL
LIN {X 0,Y 204.475,Z 146.474,A -85,B 0,C 180,E1 9203.562,E2 9203.562} C_VEL
LIN {X 0,Y 203.602,Z 142.985,A -85,B 0,C 180,E1 9201.914,E2 9201.914} C_VEL
LIN {X 0,Y 201.393,Z 138.951,A -85,B 0,C 180,E1 9198.226,E2 9198.226} C_VEL
LIN {X 0,Y 197.669,Z 134.115,A -85,B 0,C 180,E1 9188.142,E2 9188.142} C_VEL
LIN {X 0,Y 197.335,Z 134.07,A -85,B 0,C 180,E1 9183.776,E2 9183.776} C_VEL
LIN {X 0,Y 199.337,Z 138.456,A -85,B 0,C 180,E1 9173.375,E2 9173.375} C_VEL
LIN {X 0,Y 201.172,Z 142.501,A -85,B 0,C 180,E1 9169.113,E2 9169.113} C_VEL
LIN {X 0,Y 201.926,Z 144.104,A -85,B 0,C 180,E1 9167.706,E2 9167.706} C_VEL
LIN {X 0,Y 204.015,Z 148.299,A -85,B 0,C 180,E1 9164.362,E2 9164.362} C_VEL
LIN {X 0,Y 206.289,Z 153.414,A -85,B 0,C 180,E1 9161.049,E2 9161.049} C_VEL
LIN {X 0,Y 209.008,Z 160.048,A -85,B 0,C 180,E1 9157.402,E2 9157.402} C_VEL
LIN {X 0,Y 212.3,Z 168.927,A -85,B 0,C 180,E1 9153.421,E2 9153.421} C_VEL
LIN {X 0,Y 215.443,Z 179.222,A -85,B 0,C 180,E1 9149.611,E2 9149.611} C_VEL
LIN {X 0,Y 218.189,Z 190.887,A -85,B 0,C 180,E1 9146.036,E2 9146.036} C_VEL
LIN {X 0,Y 218.473,Z 193.22,A -85,B 0,C 180,E1 9145.46,E2 9145.46} C_VEL
LIN {X 0,Y 213.565,Z 227.254,A -85,B 0,C 180,E1 9140.475,E2 9140.475} C_VEL
LIN {X 0,Y 214.124,Z 234.856,A -85,B 0,C 180,E1 9139.935,E2 9139.935} C_VEL
LIN {X 0,Y 208.85,Z 318.516,A -85,B 0,C 180,E1 9137.375,E2 9137.375} C_VEL
LIN {X 0,Y 207.794,Z 344.313,A -85,B 0,C 180,E1 9136.296,E2 9136.296} C_VEL
LIN {X 0,Y 206.256,Z 358.836,A -85,B 0,C 180,E1 9135.246,E2 9135.246} C_VEL
LIN {X 0,Y 203.761,Z 372.703,A -85,B 0,C 180,E1 9133.776,E2 9133.776} C_VEL
LIN {X 0,Y 200.529,Z 385.563,A -85,B 0,C 180,E1 9131.92,E2 9131.92} C_VEL
LIN {X 0,Y 196.785,Z 397.339,A -85,B 0,C 180,E1 9129.663,E2 9129.663} C_VEL
LIN {X 0,Y 192.286,Z 408.861,A -85,B 0,C 180,E1 9126.722,E2 9126.722} C_VEL
LIN {X 0,Y 187.992,Z 418.124,A -85,B 0,C 180,E1 9123.579,E2 9123.579} C_VEL
LIN {X 0,Y 183.815,Z 426.041,A -85,B 0,C 180,E1 9120.025,E2 9120.025} C_VEL
LIN {X 0,Y 179.673,Z 432.953,A -85,B 0,C 180,E1 9115.722,E2 9115.722} C_VEL
LIN {X 0,Y 176.165,Z 438.059,A -85,B 0,C 180,E1 9110.948,E2 9110.948} C_VEL
LIN {X 0,Y 173.645,Z 441.124,A -85,B 0,C 180,E1 9106.042,E2 9106.042} C_VEL
LIN {X 0,Y 172.16,Z 442.329,A -85,B 0,C 180,E1 9101.386,E2 9101.386} C_VEL
LIN {X 0,Y 171.449,Z 441.883,A -85,B 0,C 180,E1 9096.359,E2 9096.359} C_VEL
LIN {X 0,Y 171.602,Z 439.628,A -85,B 0,C 180,E1 9091.333,E2 9091.333} C_VEL
LIN {X 0,Y 172.524,Z 435.857,A -85,B 0,C 180,E1 9086.675,E2 9086.675} C_VEL
LIN {X 0,Y 174.208,Z 430.29,A -85,B 0,C 180,E1 9082.08,E2 9082.08} C_VEL
LIN {X 0,Y 176.67,Z 422.591,A -85,B 0,C 180,E1 9077.579,E2 9077.579} C_VEL
LIN {X 0,Y 179.39,Z 413.923,A -85,B 0,C 180,E1 9073.816,E2 9073.816} C_VEL
LIN {X 0,Y 180.008,Z 411.341,A -85,B 0,C 180,E1 9072.822,E2 9072.822} C_VEL
LIN {X 0,Y 179.319,Z 411.684,A -85,B 0,C 180,E1 9072.223,E2 9072.223} C_VEL
LIN {X 0,Y 175.993,Z 421.806,A -85,B 0,C 180,E1 9067.624,E2 9067.624} C_VEL
LIN {X 0,Y 173.599,Z 429.649,A -85,B 0,C 180,E1 9062.932,E2 9062.932} C_VEL
LIN {X 0,Y 171.991,Z 436.106,A -85,B 0,C 180,E1 9057.665,E2 9057.665} C_VEL
LIN {X 0,Y 171.409,Z 440.502,A -85,B 0,C 180,E1 9052.497,E2 9052.497} C_VEL
LIN {X 0,Y 171.82,Z 443.244,A -85,B 0,C 180,E1 9047.088,E2 9047.088} C_VEL
LIN {X 0,Y 173.442,Z 444.298,A -85,B 0,C 180,E1 9041.457,E2 9041.457} C_VEL
LIN {X 0,Y 176.195,Z 443.454,A -85,B 0,C 180,E1 9036.17,E2 9036.17} C_VEL
LIN {X 0,Y 180.437,Z 440.695,A -85,B 0,C 180,E1 9030.803,E2 9030.803} C_VEL
LIN {X 0,Y 185.337,Z 436.479,A -85,B 0,C 180,E1 9026.256,E2 9026.256} C_VEL
LIN {X 0,Y 191.755,Z 429.923,A -85,B 0,C 180,E1 9021.632,E2 9021.632} C_VEL
LIN {X 0,Y 198.432,Z 422.137,A -85,B 0,C 180,E1 9017.758,E2 9017.758} C_VEL
LIN {X 0,Y 205.773,Z 412.186,A -85,B 0,C 180,E1 9014.178,E2 9014.178} C_VEL
LIN {X 0,Y 213.22,Z 400.647,A -85,B 0,C 180,E1 9011.085,E2 9011.085} C_VEL
LIN {X 0,Y 219.904,Z 388.495,A -85,B 0,C 180,E1 9008.63,E2 9008.63} C_VEL
LIN {X 0,Y 226.413,Z 374.498,A -85,B 0,C 180,E1 9006.468,E2 9006.468} C_VEL
LIN {X 0,Y 231.787,Z 360.374,A -85,B 0,C 180,E1 9004.81,E2 9004.81} C_VEL
LIN {X 0,Y 236.855,Z 343.347,A -85,B 0,C 180,E1 9003.322,E2 9003.322} C_VEL
LIN {X 0,Y 240.378,Z 327.049,A -85,B 0,C 180,E1 9002.304,E2 9002.304} C_VEL
LIN {X 0,Y 243.158,Z 306.656,A -85,B 0,C 180,E1 9001.475,E2 9001.475} C_VEL
LIN {X 0,Y 251.027,Z 242.349,A -85,B 0,C 180,E1 8999.446,E2 8999.446} C_VEL
LIN {X 0,Y 251.151,Z 228.408,A -85,B 0,C 180,E1 8997.998,E2 8997.998} C_VEL
LIN {X 0,Y 249.146,Z 222.373,A -85,B 0,C 180,E1 8995.685,E2 8995.685} C_VEL
LIN {X 0,Y 247.816,Z 218.569,A -85,B 0,C 180,E1 8993.863,E2 8993.863} C_VEL
LIN {X 0,Y 246.12,Z 213.807,A -85,B 0,C 180,E1 8990.822,E2 8990.822} C_VEL
LIN {X 0,Y 244.949,Z 210.201,A -85,B 0,C 180,E1 8986.787,E2 8986.787} C_VEL
LIN {X 0,Y 245.013,Z 209.472,A -85,B 0,C 180,E1 8982.669,E2 8982.669} C_VEL
LIN {X 0,Y 246.556,Z 211.255,A -85,B 0,C 180,E1 8978.344,E2 8978.344} C_VEL
LIN {X 0,Y 248.492,Z 214.423,A -85,B 0,C 180,E1 8975.39,E2 8975.39} C_VEL
LIN {X 0,Y 250.911,Z 218.978,A -85,B 0,C 180,E1 8972.661,E2 8972.661} C_VEL
LIN {X 0,Y 252.746,Z 222.711,A -85,B 0,C 180,E1 8970.941,E2 8970.941} C_VEL
LIN {X 0,Y 253.001,Z 224.692,A -85,B 0,C 180,E1 8970.582,E2 8970.582} C_VEL
LIN {X 0,Y 252.703,Z 228.033,A -85,B 0,C 180,E1 8970.443,E2 8970.443} C_VEL
LIN {X 0,Y 251.649,Z 233.026,A -85,B 0,C 180,E1 8970.618,E2 8970.618} C_VEL
LIN {X 0,Y 249.109,Z 242.877,A -85,B 0,C 180,E1 8971.279,E2 8971.279} C_VEL
LIN {X 0,Y 248.558,Z 246.292,A -85,B 0,C 180,E1 8971.295,E2 8971.295} C_VEL
LIN {X 0,Y 238.401,Z 335.366,A -85,B 0,C 180,E1 8968.855,E2 8968.855} C_VEL
LIN {X 0,Y 234.577,Z 354.021,A -85,B 0,C 180,E1 8968.084,E2 8968.084} C_VEL
LIN {X 0,Y 229.778,Z 370.507,A -85,B 0,C 180,E1 8967.123,E2 8967.123} C_VEL
LIN {X 0,Y 223.62,Z 386.847,A -85,B 0,C 180,E1 8965.812,E2 8965.812} C_VEL
LIN {X 0,Y 216.529,Z 402.277,A -85,B 0,C 180,E1 8964.115,E2 8964.115} C_VEL
LIN {X 0,Y 208.439,Z 417.273,A -85,B 0,C 180,E1 8961.879,E2 8961.879} C_VEL
LIN {X 0,Y 199.836,Z 431.282,A -85,B 0,C 180,E1 8959.072,E2 8959.072} C_VEL
LIN {X 0,Y 191.317,Z 443.654,A -85,B 0,C 180,E1 8955.726,E2 8955.726} C_VEL
LIN {X 0,Y 183.149,Z 454.598,A -85,B 0,C 180,E1 8951.764,E2 8951.764} C_VEL
LIN {X 0,Y 175.673,Z 464.211,A -85,B 0,C 180,E1 8947.109,E2 8947.109} C_VEL
LIN {X 0,Y 169.289,Z 472.418,A -85,B 0,C 180,E1 8941.715,E2 8941.715} C_VEL
LIN {X 0,Y 164.451,Z 479.148,A -85,B 0,C 180,E1 8935.577,E2 8935.577} C_VEL
LIN {X 0,Y 161.589,Z 484.21,A -85,B 0,C 180,E1 8928.791,E2 8928.791} C_VEL
LIN {X 0,Y 161.001,Z 487.405,A -85,B 0,C 180,E1 8921.828,E2 8921.828} C_VEL
LIN {X 0,Y 162.211,Z 488.664,A -85,B 0,C 180,E1 8915.308,E2 8915.308} C_VEL
LIN {X 0,Y 163.499,Z 488.402,A -85,B 0,C 180,E1 8910.703,E2 8910.703} C_VEL
LIN {X 0,Y 163.39,Z 488.196,A -85,B 0,C 180,E1 8908.6,E2 8908.6} C_VEL
LIN {X 0,Y 162.049,Z 487.959,A -85,B 0,C 180,E1 8903.982,E2 8903.982} C_VEL
LIN {X 0,Y 161.106,Z 485.874,A -85,B 0,C 180,E1 8898.548,E2 8898.548} C_VEL
LIN {X 0,Y 161.264,Z 482.253,A -85,B 0,C 180,E1 8893.432,E2 8893.432} C_VEL
LIN {X 0,Y 162.744,Z 476.421,A -85,B 0,C 180,E1 8887.993,E2 8887.993} C_VEL
LIN {X 0,Y 165.363,Z 468.866,A -85,B 0,C 180,E1 8883.036,E2 8883.036} C_VEL
LIN {X 0,Y 168.532,Z 460.487,A -85,B 0,C 180,E1 8878.929,E2 8878.929} C_VEL
LIN {X 0,Y 172.331,Z 450.404,A -85,B 0,C 180,E1 8875.149,E2 8875.149} C_VEL
LIN {X 0,Y 176.615,Z 438.089,A -85,B 0,C 180,E1 8871.695,E2 8871.695} C_VEL
LIN {X 0,Y 180.543,Z 425.103,A -85,B 0,C 180,E1 8868.989,E2 8868.989} C_VEL
LIN {X 0,Y 183.806,Z 411.995,A -85,B 0,C 180,E1 8866.95,E2 8866.95} C_VEL
LIN {X 0,Y 186.223,Z 400.354,A -85,B 0,C 180,E1 8865.545,E2 8865.545} C_VEL
LIN {X 0,Y 190.693,Z 384.304,A -85,B 0,C 180,E1 8863.351,E2 8863.351} C_VEL
LIN {X 0,Y 194.54,Z 367.464,A -85,B 0,C 180,E1 8861.666,E2 8861.666} C_VEL
LIN {X 0,Y 197.556,Z 349.385,A -85,B 0,C 180,E1 8860.39,E2 8860.39} C_VEL
LIN {X 0,Y 199.339,Z 331.218,A -85,B 0,C 180,E1 8859.555,E2 8859.555} C_VEL
LIN {X 0,Y 209.04,Z 192.631,A -85,B 0,C 180,E1 8855.084,E2 8855.084} C_VEL
LIN {X 0,Y 209.529,Z 189.353,A -85,B 0,C 180,E1 8854.821,E2 8854.821} C_VEL
LIN {X 0,Y 207.195,Z 178.812,A -85,B 0,C 180,E1 8852.02,E2 8852.02} C_VEL
LIN {X 0,Y 203.712,Z 164.43,A -85,B 0,C 180,E1 8847.272,E2 8847.272} C_VEL
LIN {X 0,Y 201.144,Z 152.87,A -85,B 0,C 180,E1 8842.581,E2 8842.581} C_VEL
LIN {X 0,Y 200.38,Z 149.868,A -85,B 0,C 180,E1 8841.055,E2 8841.055} C_VEL
LIN {X 0,Y 198.439,Z 146.313,A -85,B 0,C 180,E1 8837.778,E2 8837.778} C_VEL
LIN {X 0,Y 194.919,Z 141.608,A -85,B 0,C 180,E1 8827.96,E2 8827.96} C_VEL
LIN {X 0,Y 194.412,Z 141.526,A -85,B 0,C 180,E1 8823.833,E2 8823.833} C_VEL
LIN {X 0,Y 196.043,Z 145.573,A -85,B 0,C 180,E1 8813.851,E2 8813.851} C_VEL
LIN {X 0,Y 197.764,Z 149.617,A -85,B 0,C 180,E1 8809.513,E2 8809.513} C_VEL
LIN {X 0,Y 200.345,Z 155.094,A -85,B 0,C 180,E1 8804.958,E2 8804.958} C_VEL
LIN {X 0,Y 203.016,Z 161.669,A -85,B 0,C 180,E1 8800.582,E2 8800.582} C_VEL
LIN {X 0,Y 206.126,Z 170.146,A -85,B 0,C 180,E1 8796.258,E2 8796.258} C_VEL
LIN {X 0,Y 208.955,Z 178.744,A -85,B 0,C 180,E1 8792.653,E2 8792.653} C_VEL
LIN {X 0,Y 211.602,Z 189.124,A -85,B 0,C 180,E1 8788.999,E2 8788.999} C_VEL
LIN {X 0,Y 213.034,Z 196.715,A -85,B 0,C 180,E1 8786.764,E2 8786.764} C_VEL
LIN {X 0,Y 208.186,Z 228.204,A -85,B 0,C 180,E1 8782.102,E2 8782.102} C_VEL
LIN {X 0,Y 208.717,Z 236.082,A -85,B 0,C 180,E1 8781.52,E2 8781.52} C_VEL
LIN {X 0,Y 203.237,Z 318.972,A -85,B 0,C 180,E1 8778.955,E2 8778.955} C_VEL
LIN {X 0,Y 202.061,Z 345.346,A -85,B 0,C 180,E1 8777.832,E2 8777.832} C_VEL
LIN {X 0,Y 200.407,Z 360.037,A -85,B 0,C 180,E1 8776.749,E2 8776.749} C_VEL
LIN {X 0,Y 197.776,Z 373.878,A -85,B 0,C 180,E1 8775.255,E2 8775.255} C_VEL
LIN {X 0,Y 194.378,Z 386.719,A -85,B 0,C 180,E1 8773.366,E2 8773.366} C_VEL
LIN {X 0,Y 190.38,Z 398.647,A -85,B 0,C 180,E1 8771.029,E2 8771.029} C_VEL
LIN {X 0,Y 185.488,Z 410.484,A -85,B 0,C 180,E1 8767.913,E2 8767.913} C_VEL
LIN {X 0,Y 180.587,Z 420.37,A -85,B 0,C 180,E1 8764.381,E2 8764.381} C_VEL
LIN {X 0,Y 175.898,Z 428.545,A -85,B 0,C 180,E1 8760.388,E2 8760.388} C_VEL
LIN {X 0,Y 171.925,Z 434.663,A -85,B 0,C 180,E1 8756.228,E2 8756.228} C_VEL
LIN {X 0,Y 168.499,Z 439.312,A -85,B 0,C 180,E1 8751.583,E2 8751.583} C_VEL
LIN {X 0,Y 165.83,Z 442.302,A -85,B 0,C 180,E1 8746.459,E2 8746.459} C_VEL
LIN {X 0,Y 164.179,Z 443.449,A -85,B 0,C 180,E1 8741.235,E2 8741.235} C_VEL
LIN {X 0,Y 163.5,Z 442.825,A -85,B 0,C 180,E1 8735.965,E2 8735.965} C_VEL
LIN {X 0,Y 163.747,Z 440.406,A -85,B 0,C 180,E1 8730.697,E2 8730.697} C_VEL
LIN {X 0,Y 164.916,Z 436.073,A -85,B 0,C 180,E1 8725.477,E2 8725.477} C_VEL
LIN {X 0,Y 166.685,Z 430.622,A -85,B 0,C 180,E1 8721.025,E2 8721.025} C_VEL
LIN {X 0,Y 169.173,Z 423.341,A -85,B 0,C 180,E1 8716.671,E2 8716.671} C_VEL
LIN {X 0,Y 171.888,Z 414.793,A -85,B 0,C 180,E1 8712.816,E2 8712.816} C_VEL
LIN {X 0,Y 171.065,Z 414.592,A -85,B 0,C 180,E1 8712.186,E2 8712.186} C_VEL
LIN {X 0,Y 167.618,Z 424.502,A -85,B 0,C 180,E1 8707.184,E2 8707.184} C_VEL
LIN {X 0,Y 165.157,Z 432.536,A -85,B 0,C 180,E1 8701.82,E2 8701.82} C_VEL
LIN {X 0,Y 163.84,Z 438.131,A -85,B 0,C 180,E1 8696.683,E2 8696.683} C_VEL
LIN {X 0,Y 163.472,Z 442.391,A -85,B 0,C 180,E1 8690.948,E2 8690.948} C_VEL
LIN {X 0,Y 164.211,Z 444.773,A -85,B 0,C 180,E1 8685.431,E2 8685.431} C_VEL
LIN {X 0,Y 166.248,Z 445.441,A -85,B 0,C 180,E1 8679.608,E2 8679.608} C_VEL
LIN {X 0,Y 169.74,Z 444.261,A -85,B 0,C 180,E1 8673.84,E2 8673.84} C_VEL
LIN {X 0,Y 174.331,Z 441.308,A -85,B 0,C 180,E1 8668.652,E2 8668.652} C_VEL
LIN {X 0,Y 180.497,Z 436.231,A -85,B 0,C 180,E1 8663.507,E2 8663.507} C_VEL
LIN {X 0,Y 186.801,Z 430.117,A -85,B 0,C 180,E1 8659.382,E2 8659.382} C_VEL
LIN {X 0,Y 194.025,Z 421.958,A -85,B 0,C 180,E1 8655.489,E2 8655.489} C_VEL
LIN {X 0,Y 201.709,Z 412.082,A -85,B 0,C 180,E1 8652.017,E2 8652.017} C_VEL
LIN {X 0,Y 208.708,Z 401.713,A -85,B 0,C 180,E1 8649.282,E2 8649.282} C_VEL
LIN {X 0,Y 216.016,Z 388.975,A -85,B 0,C 180,E1 8646.739,E2 8646.739} C_VEL
LIN {X 0,Y 222.743,Z 375.177,A -85,B 0,C 180,E1 8644.635,E2 8644.635} C_VEL
LIN {X 0,Y 228.577,Z 360.439,A -85,B 0,C 180,E1 8642.94,E2 8642.94} C_VEL
LIN {X 0,Y 233.642,Z 344.039,A -85,B 0,C 180,E1 8641.539,E2 8641.539} C_VEL
LIN {X 0,Y 237.3,Z 327.656,A -85,B 0,C 180,E1 8640.536,E2 8640.536} C_VEL
LIN {X 0,Y 240.216,Z 306.928,A -85,B 0,C 180,E1 8639.71,E2 8639.71} C_VEL
LIN {X 0,Y 248.179,Z 244.226,A -85,B 0,C 180,E1 8637.765,E2 8637.765} C_VEL
LIN {X 0,Y 248.462,Z 233.777,A -85,B 0,C 180,E1 8636.655,E2 8636.655} C_VEL
LIN {X 0,Y 246.825,Z 228.374,A -85,B 0,C 180,E1 8634.48,E2 8634.48} C_VEL
LIN {X 0,Y 245.694,Z 224.888,A -85,B 0,C 180,E1 8632.635,E2 8632.635} C_VEL
LIN {X 0,Y 244.546,Z 221.156,A -85,B 0,C 180,E1 8630.112,E2 8630.112} C_VEL
LIN {X 0,Y 243.618,Z 217.859,A -85,B 0,C 180,E1 8625.987,E2 8625.987} C_VEL
LIN {X 0,Y 243.861,Z 217.434,A -85,B 0,C 180,E1 8622.338,E2 8622.338} C_VEL
LIN {X 0,Y 245.529,Z 219.471,A -85,B 0,C 180,E1 8617.998,E2 8617.998} C_VEL
LIN {X 0,Y 247.394,Z 223.133,A -85,B 0,C 180,E1 8615.145,E2 8615.145} C_VEL
LIN {X 0,Y 249.239,Z 226.739,A -85,B 0,C 180,E1 8613.044,E2 8613.044} C_VEL
LIN {X 0,Y 250.475,Z 229.801,A -85,B 0,C 180,E1 8611.729,E2 8611.729} C_VEL
LIN {X 0,Y 248.558,Z 246.292,A -85,B 0,C 180,E1 8611.295,E2 8611.295} C_VEL
LIN {X 0,Y 247.358,Z 253.965,A -85,B 0,C 180,E1 8611.312,E2 8611.312} C_VEL
LIN {X 0,Y 243.031,Z 274.448,A -85,B 0,C 180,E1 8612.164,E2 8612.164} C_VEL
LIN {X 0,Y 242.028,Z 281.031,A -85,B 0,C 180,E1 8612.159,E2 8612.159} C_VEL
LIN {X 0,Y 235.511,Z 335.109,A -85,B 0,C 180,E1 8610.669,E2 8610.669} C_VEL
LIN {X 0,Y 231.589,Z 353.52,A -85,B 0,C 180,E1 8609.926,E2 8609.926} C_VEL
LIN {X 0,Y 226.407,Z 370.52,A -85,B 0,C 180,E1 8608.955,E2 8608.955} C_VEL
LIN {X 0,Y 220.055,Z 386.519,A -85,B 0,C 180,E1 8607.687,E2 8607.687} C_VEL
LIN {X 0,Y 212.381,Z 402.415,A -85,B 0,C 180,E1 8605.955,E2 8605.955} C_VEL
LIN {X 0,Y 203.963,Z 417.295,A -85,B 0,C 180,E1 8603.749,E2 8603.749} C_VEL
LIN {X 0,Y 195.326,Z 430.548,A -85,B 0,C 180,E1 8601.087,E2 8601.087} C_VEL
LIN {X 0,Y 186.361,Z 442.788,A -85,B 0,C 180,E1 8597.767,E2 8597.767} C_VEL
LIN {X 0,Y 177.158,Z 454.35,A -85,B 0,C 180,E1 8593.518,E2 8593.518} C_VEL
LIN {X 0,Y 169.08,Z 463.92,A -85,B 0,C 180,E1 8588.687,E2 8588.687} C_VEL
LIN {X 0,Y 162.008,Z 472.187,A -85,B 0,C 180,E1 8582.898,E2 8582.898} C_VEL
LIN {X 0,Y 156.838,Z 478.611,A -85,B 0,C 180,E1 8576.506,E2 8576.506} C_VEL
LIN {X 0,Y 153.722,Z 483.461,A -85,B 0,C 180,E1 8569.376,E2 8569.376} C_VEL
LIN {X 0,Y 153.032,Z 486.441,A -85,B 0,C 180,E1 8562.071,E2 8562.071} C_VEL
LIN {X 0,Y 154.28,Z 487.496,A -85,B 0,C 180,E1 8555.208,E2 8555.208} C_VEL
LIN {X 0,Y 155.583,Z 487.113,A -85,B 0,C 180,E1 8550.739,E2 8550.739} C_VEL
LIN {X 0,Y 155.516,Z 487.019,A -85,B 0,C 180,E1 8548.898,E2 8548.898} C_VEL
LIN {X 0,Y 154.092,Z 486.907,A -85,B 0,C 180,E1 8544.044,E2 8544.044} C_VEL
LIN {X 0,Y 153.122,Z 485.024,A -85,B 0,C 180,E1 8538.368,E2 8538.368} C_VEL
LIN {X 0,Y 153.399,Z 481.237,A -85,B 0,C 180,E1 8532.556,E2 8532.556} C_VEL
LIN {X 0,Y 155.136,Z 475.45,A -85,B 0,C 180,E1 8526.853,E2 8526.853} C_VEL
LIN {X 0,Y 158.052,Z 467.955,A -85,B 0,C 180,E1 8521.679,E2 8521.679} C_VEL
LIN {X 0,Y 161.71,Z 459.229,A -85,B 0,C 180,E1 8517.233,E2 8517.233} C_VEL
LIN {X 0,Y 166.047,Z 448.696,A -85,B 0,C 180,E1 8513.212,E2 8513.212} C_VEL
LIN {X 0,Y 170.515,Z 436.838,A -85,B 0,C 180,E1 8509.837,E2 8509.837} C_VEL
LIN {X 0,Y 174.735,Z 423.824,A -85,B 0,C 180,E1 8507.088,E2 8507.088} C_VEL
LIN {X 0,Y 178.221,Z 410.671,A -85,B 0,C 180,E1 8505.022,E2 8505.022} C_VEL
LIN {X 0,Y 181.045,Z 396.66,A -85,B 0,C 180,E1 8503.433,E2 8503.433} C_VEL
LIN {X 0,Y 182.425,Z 389.268,A -85,B 0,C 180,E1 8502.744,E2 8502.744} C_VEL
LIN {X 0,Y 186.75,Z 372.311,A -85,B 0,C 180,E1 8500.817,E2 8500.817} C_VEL
LIN {X 0,Y 190.211,Z 354.581,A -85,B 0,C 180,E1 8499.377,E2 8499.377} C_VEL
LIN {X 0,Y 192.422,Z 336.603,A -85,B 0,C 180,E1 8498.394,E2 8498.394} C_VEL
LIN {X 0,Y 202.035,Z 205.784,A -85,B 0,C 180,E1 8494.03,E2 8494.03} C_VEL
LIN {X 0,Y 204.743,Z 192.456,A -85,B 0,C 180,E1 8493.116,E2 8493.116} C_VEL
LIN {X 0,Y 202.861,Z 183.382,A -85,B 0,C 180,E1 8490.59,E2 8490.59} C_VEL
LIN {X 0,Y 199.927,Z 170.021,A -85,B 0,C 180,E1 8486.03,E2 8486.03} C_VEL
LIN {X 0,Y 197.841,Z 159.114,A -85,B 0,C 180,E1 8481.494,E2 8481.494} C_VEL
LIN {X 0,Y 197.309,Z 156.877,A -85,B 0,C 180,E1 8480.311,E2 8480.311} C_VEL
LIN {X 0,Y 195.72,Z 153.802,A -85,B 0,C 180,E1 8477.542,E2 8477.542} C_VEL
LIN {X 0,Y 192.291,Z 149.143,A -85,B 0,C 180,E1 8467.769,E2 8467.769} C_VEL
LIN {X 0,Y 191.822,Z 149.109,A -85,B 0,C 180,E1 8463.885,E2 8463.885} C_VEL
LIN {X 0,Y 193.176,Z 153.156,A -85,B 0,C 180,E1 8454.058,E2 8454.058} C_VEL
LIN {X 0,Y 195.028,Z 157.753,A -85,B 0,C 180,E1 8449.065,E2 8449.065} C_VEL
LIN {X 0,Y 196.85,Z 162.326,A -85,B 0,C 180,E1 8445.287,E2 8445.287} C_VEL
LIN {X 0,Y 199.164,Z 168.286,A -85,B 0,C 180,E1 8441.258,E2 8441.258} C_VEL
LIN {X 0,Y 202.178,Z 177.088,A -85,B 0,C 180,E1 8436.694,E2 8436.694} C_VEL
LIN {X 0,Y 204.858,Z 186.617,A -85,B 0,C 180,E1 8432.69,E2 8432.69} C_VEL
LIN {X 0,Y 207.22,Z 197.129,A -85,B 0,C 180,E1 8429.077,E2 8429.077} C_VEL
LIN {X 0,Y 207.683,Z 200.437,A -85,B 0,C 180,E1 8428.103,E2 8428.103} C_VEL
LIN {X 0,Y 202.996,Z 229.318,A -85,B 0,C 180,E1 8423.799,E2 8423.799} C_VEL
LIN {X 0,Y 203.485,Z 237.19,A -85,B 0,C 180,E1 8423.191,E2 8423.191} C_VEL
LIN {X 0,Y 197.788,Z 319.428,A -85,B 0,C 180,E1 8420.624,E2 8420.624} C_VEL
LIN {X 0,Y 196.471,Z 346.521,A -85,B 0,C 180,E1 8419.448,E2 8419.448} C_VEL
LIN {X 0,Y 194.706,Z 361.248,A -85,B 0,C 180,E1 8418.342,E2 8418.342} C_VEL
LIN {X 0,Y 191.679,Z 376.15,A -85,B 0,C 180,E1 8416.687,E2 8416.687} C_VEL
LIN {X 0,Y 187.856,Z 389.451,A -85,B 0,C 180,E1 8414.629,E2 8414.629} C_VEL
LIN {X 0,Y 183.648,Z 401.027,A -85,B 0,C 180,E1 8412.23,E2 8412.23} C_VEL
LIN {X 0,Y 178.772,Z 412.078,A -85,B 0,C 180,E1 8409.194,E2 8409.194} C_VEL
LIN {X 0,Y 173.621,Z 421.87,A -85,B 0,C 180,E1 8405.563,E2 8405.563} C_VEL
LIN {X 0,Y 168.567,Z 430.121,A -85,B 0,C 180,E1 8401.333,E2 8401.333} C_VEL
LIN {X 0,Y 164.19,Z 436.359,A -85,B 0,C 180,E1 8396.781,E2 8396.781} C_VEL
LIN {X 0,Y 160.628,Z 440.795,A -85,B 0,C 180,E1 8391.927,E2 8391.927} C_VEL
LIN {X 0,Y 157.875,Z 443.621,A -85,B 0,C 180,E1 8386.555,E2 8386.555} C_VEL
LIN {X 0,Y 156.127,Z 444.583,A -85,B 0,C 180,E1 8380.7,E2 8380.7} C_VEL
LIN {X 0,Y 155.547,Z 443.54,A -85,B 0,C 180,E1 8374.892,E2 8374.892} C_VEL
LIN {X 0,Y 155.986,Z 440.797,A -85,B 0,C 180,E1 8369.501,E2 8369.501} C_VEL
LIN {X 0,Y 157.376,Z 436.232,A -85,B 0,C 180,E1 8364.163,E2 8364.163} C_VEL
LIN {X 0,Y 159.596,Z 429.937,A -85,B 0,C 180,E1 8359.164,E2 8359.164} C_VEL
LIN {X 0,Y 162.691,Z 421.366,A -85,B 0,C 180,E1 8354.309,E2 8354.309} C_VEL
LIN {X 0,Y 163.714,Z 418.048,A -85,B 0,C 180,E1 8352.767,E2 8352.767} C_VEL
LIN {X 0,Y 162.692,Z 417.631,A -85,B 0,C 180,E1 8352.009,E2 8352.009} C_VEL
LIN {X 0,Y 159.026,Z 427.802,A -85,B 0,C 180,E1 8346.27,E2 8346.27} C_VEL
LIN {X 0,Y 156.828,Z 434.958,A -85,B 0,C 180,E1 8340.863,E2 8340.863} C_VEL
LIN {X 0,Y 155.67,Z 440.462,A -85,B 0,C 180,E1 8335.132,E2 8335.132} C_VEL
LIN {X 0,Y 155.633,Z 444.193,A -85,B 0,C 180,E1 8329.297,E2 8329.297} C_VEL
LIN {X 0,Y 156.919,Z 446.303,A -85,B 0,C 180,E1 8322.984,E2 8322.984} C_VEL
LIN {X 0,Y 159.59,Z 446.543,A -85,B 0,C 180,E1 8316.975,E2 8316.975} C_VEL
LIN {X 0,Y 163.678,Z 444.909,A -85,B 0,C 180,E1 8311.213,E2 8311.213} C_VEL
LIN {X 0,Y 168.992,Z 441.591,A -85,B 0,C 180,E1 8305.927,E2 8305.927} C_VEL
LIN {X 0,Y 175.483,Z 436.456,A -85,B 0,C 180,E1 8301.037,E2 8301.037} C_VEL
LIN {X 0,Y 183.123,Z 429.283,A -85,B 0,C 180,E1 8296.495,E2 8296.495} C_VEL
LIN {X 0,Y 190.916,Z 420.828,A -85,B 0,C 180,E1 8292.707,E2 8292.707} C_VEL
LIN {X 0,Y 198.694,Z 410.963,A -85,B 0,C 180,E1 8289.488,E2 8289.488} C_VEL
LIN {X 0,Y 206.837,Z 399.08,A -85,B 0,C 180,E1 8286.581,E2 8286.581} C_VEL
LIN {X 0,Y 214.079,Z 386.631,A -85,B 0,C 180,E1 8284.286,E2 8284.286} C_VEL
LIN {X 0,Y 220.792,Z 372.673,A -85,B 0,C 180,E1 8282.336,E2 8282.336} C_VEL
LIN {X 0,Y 226.987,Z 356.83,A -85,B 0,C 180,E1 8280.671,E2 8280.671} C_VEL
LIN {X 0,Y 231.734,Z 340.893,A -85,B 0,C 180,E1 8279.44,E2 8279.44} C_VEL
LIN {X 0,Y 235.376,Z 323.687,A -85,B 0,C 180,E1 8278.498,E2 8278.498} C_VEL
LIN {X 0,Y 240.683,Z 284.122,A -85,B 0,C 180,E1 8277.191,E2 8277.191} C_VEL
LIN {X 0,Y 245.649,Z 246.048,A -85,B 0,C 180,E1 8276.033,E2 8276.033} C_VEL
LIN {X 0,Y 245.924,Z 239.159,A -85,B 0,C 180,E1 8275.296,E2 8275.296} C_VEL
LIN {X 0,Y 244.323,Z 233.206,A -85,B 0,C 180,E1 8272.594,E2 8272.594} C_VEL
LIN {X 0,Y 243.114,Z 228.823,A -85,B 0,C 180,E1 8269.695,E2 8269.695} C_VEL
LIN {X 0,Y 242.371,Z 225.726,A -85,B 0,C 180,E1 8265.804,E2 8265.804} C_VEL
LIN {X 0,Y 242.616,Z 225.32,A -85,B 0,C 180,E1 8262.492,E2 8262.492} C_VEL
LIN {X 0,Y 244.164,Z 227.309,A -85,B 0,C 180,E1 8258.248,E2 8258.248} C_VEL
LIN {X 0,Y 245.962,Z 231.07,A -85,B 0,C 180,E1 8255.376,E2 8255.376} C_VEL
LIN {X 0,Y 247.613,Z 234.693,A -85,B 0,C 180,E1 8253.371,E2 8253.371} C_VEL
LIN {X 0,Y 242.028,Z 281.031,A -85,B 0,C 180,E1 8252.159,E2 8252.159} C_VEL
LIN {X 0,Y 240.831,Z 288.703,A -85,B 0,C 180,E1 8252.182,E2 8252.182} C_VEL
LIN {X 0,Y 236.581,Z 309.186,A -85,B 0,C 180,E1 8253.08,E2 8253.08} C_VEL
LIN {X 0,Y 235.571,Z 315.768,A -85,B 0,C 180,E1 8253.078,E2 8253.078} C_VEL
LIN {X 0,Y 232.346,Z 338.214,A -85,B 0,C 180,E1 8252.42,E2 8252.42} C_VEL
LIN {X 0,Y 228.242,Z 355.369,A -85,B 0,C 180,E1 8251.707,E2 8251.707} C_VEL
LIN {X 0,Y 222.45,Z 372.718,A -85,B 0,C 180,E1 8250.692,E2 8250.692} C_VEL
LIN {X 0,Y 215.537,Z 388.991,A -85,B 0,C 180,E1 8249.377,E2 8249.377} C_VEL
LIN {X 0,Y 207.662,Z 404.253,A -85,B 0,C 180,E1 8247.675,E2 8247.675} C_VEL
LIN {X 0,Y 198.975,Z 418.446,A -85,B 0,C 180,E1 8245.501,E2 8245.501} C_VEL
LIN {X 0,Y 188.998,Z 432.662,A -85,B 0,C 180,E1 8242.521,E2 8242.521} C_VEL
LIN {X 0,Y 179.757,Z 444.39,A -85,B 0,C 180,E1 8239.156,E2 8239.156} C_VEL
LIN {X 0,Y 170.783,Z 454.768,A -85,B 0,C 180,E1 8235.108,E2 8235.108} C_VEL
LIN {X 0,Y 161.964,Z 464.321,A -85,B 0,C 180,E1 8229.946,E2 8229.946} C_VEL
LIN {X 0,Y 154.438,Z 472.306,A -85,B 0,C 180,E1 8223.836,E2 8223.836} C_VEL
LIN {X 0,Y 149.026,Z 478.397,A -85,B 0,C 180,E1 8217.147,E2 8217.147} C_VEL
LIN {X 0,Y 145.772,Z 482.897,A -85,B 0,C 180,E1 8209.642,E2 8209.642} C_VEL
LIN {X 0,Y 145.098,Z 485.494,A -85,B 0,C 180,E1 8201.903,E2 8201.903} C_VEL
LIN {X 0,Y 146.482,Z 486.213,A -85,B 0,C 180,E1 8194.701,E2 8194.701} C_VEL
LIN {X 0,Y 147.791,Z 485.699,A -85,B 0,C 180,E1 8190.003,E2 8190.003} C_VEL
LIN {X 0,Y 146.463,Z 485.998,A -85,B 0,C 180,E1 8185.304,E2 8185.304} C_VEL
LIN {X 0,Y 145.234,Z 484.608,A -85,B 0,C 180,E1 8179.291,E2 8179.291} C_VEL
LIN {X 0,Y 145.247,Z 481.669,A -85,B 0,C 180,E1 8173.61,E2 8173.61} C_VEL
LIN {X 0,Y 146.741,Z 476.626,A -85,B 0,C 180,E1 8167.573,E2 8167.573} C_VEL
LIN {X 0,Y 149.538,Z 469.944,A -85,B 0,C 180,E1 8162.096,E2 8162.096} C_VEL
LIN {X 0,Y 153.295,Z 461.782,A -85,B 0,C 180,E1 8157.227,E2 8157.227} C_VEL
LIN {X 0,Y 157.698,Z 452.182,A -85,B 0,C 180,E1 8152.967,E2 8152.967} C_VEL
LIN {X 0,Y 162.735,Z 440.315,A -85,B 0,C 180,E1 8149.088,E2 8149.088} C_VEL
LIN {X 0,Y 167.32,Z 428,A -85,B 0,C 180,E1 8146.122,E2 8146.122} C_VEL
LIN {X 0,Y 171.265,Z 415.48,A -85,B 0,C 180,E1 8143.868,E2 8143.868} C_VEL
LIN {X 0,Y 174.813,Z 400.994,A -85,B 0,C 180,E1 8141.97,E2 8141.97} C_VEL
LIN {X 0,Y 177.434,Z 385.352,A -85,B 0,C 180,E1 8140.584,E2 8140.584} C_VEL
LIN {X 0,Y 178.494,Z 378.522,A -85,B 0,C 180,E1 8140.104,E2 8140.104} C_VEL
LIN {X 0,Y 182.523,Z 360.802,A -85,B 0,C 180,E1 8138.437,E2 8138.437} C_VEL
LIN {X 0,Y 185.279,Z 342.981,A -85,B 0,C 180,E1 8137.273,E2 8137.273} C_VEL
LIN {X 0,Y 187.243,Z 319.87,A -85,B 0,C 180,E1 8136.353,E2 8136.353} C_VEL
LIN {X 0,Y 194.979,Z 219.054,A -85,B 0,C 180,E1 8132.938,E2 8132.938} C_VEL
LIN {X 0,Y 200.133,Z 195.559,A -85,B 0,C 180,E1 8131.341,E2 8131.341} C_VEL
LIN {X 0,Y 198.312,Z 186.343,A -85,B 0,C 180,E1 8128.577,E2 8128.577} C_VEL
LIN {X 0,Y 196.055,Z 174.913,A -85,B 0,C 180,E1 8124.479,E2 8124.479} C_VEL
LIN {X 0,Y 194.524,Z 165.473,A -85,B 0,C 180,E1 8120.458,E2 8120.458} C_VEL
LIN {X 0,Y 194.197,Z 163.852,A -85,B 0,C 180,E1 8119.552,E2 8119.552} C_VEL
LIN {X 0,Y 192.81,Z 161.124,A -85,B 0,C 180,E1 8116.881,E2 8116.881} C_VEL
LIN {X 0,Y 189.665,Z 156.68,A -85,B 0,C 180,E1 8107.573,E2 8107.573} C_VEL
LIN {X 0,Y 189.203,Z 156.773,A -85,B 0,C 180,E1 8103.635,E2 8103.635} C_VEL
LIN {X 0,Y 190.124,Z 160.36,A -85,B 0,C 180,E1 8094.568,E2 8094.568} C_VEL
LIN {X 0,Y 191.649,Z 164.92,A -85,B 0,C 180,E1 8089.478,E2 8089.478} C_VEL
LIN {X 0,Y 193.366,Z 169.544,A -85,B 0,C 180,E1 8085.628,E2 8085.628} C_VEL
LIN {X 0,Y 195.416,Z 175.166,A -85,B 0,C 180,E1 8081.813,E2 8081.813} C_VEL
LIN {X 0,Y 197.898,Z 183.37,A -85,B 0,C 180,E1 8077.419,E2 8077.419} C_VEL
LIN {X 0,Y 200.185,Z 192.246,A -85,B 0,C 180,E1 8073.606,E2 8073.606} C_VEL
LIN {X 0,Y 202.316,Z 202.405,A -85,B 0,C 180,E1 8070.055,E2 8070.055} C_VEL
LIN {X 0,Y 202.507,Z 204.266,A -85,B 0,C 180,E1 8069.514,E2 8069.514} C_VEL
LIN {X 0,Y 197.99,Z 230.396,A -85,B 0,C 180,E1 8065.587,E2 8065.587} C_VEL
LIN {X 0,Y 198.424,Z 238.449,A -85,B 0,C 180,E1 8064.945,E2 8064.945} C_VEL
LIN {X 0,Y 192.517,Z 319.891,A -85,B 0,C 180,E1 8062.386,E2 8062.386} C_VEL
LIN {X 0,Y 191.062,Z 347.55,A -85,B 0,C 180,E1 8061.166,E2 8061.166} C_VEL
LIN {X 0,Y 189.164,Z 362.464,A -85,B 0,C 180,E1 8060.029,E2 8060.029} C_VEL
LIN {X 0,Y 185.976,Z 377.337,A -85,B 0,C 180,E1 8058.353,E2 8058.353} C_VEL
LIN {X 0,Y 181.958,Z 390.617,A -85,B 0,C 180,E1 8056.264,E2 8056.264} C_VEL
LIN {X 0,Y 177.552,Z 402.128,A -85,B 0,C 180,E1 8053.837,E2 8053.837} C_VEL
LIN {X 0,Y 172.631,Z 412.762,A -85,B 0,C 180,E1 8050.876,E2 8050.876} C_VEL
LIN {X 0,Y 167.163,Z 422.632,A -85,B 0,C 180,E1 8047.161,E2 8047.161} C_VEL
LIN {X 0,Y 161.894,Z 430.791,A -85,B 0,C 180,E1 8042.918,E2 8042.918} C_VEL
LIN {X 0,Y 157.392,Z 436.895,A -85,B 0,C 180,E1 8038.45,E2 8038.45} C_VEL
LIN {X 0,Y 153.475,Z 441.534,A -85,B 0,C 180,E1 8033.412,E2 8033.412} C_VEL
LIN {X 0,Y 150.392,Z 444.511,A -85,B 0,C 180,E1 8027.804,E2 8027.804} C_VEL
LIN {X 0,Y 148.461,Z 445.644,A -85,B 0,C 180,E1 8022.048,E2 8022.048} C_VEL
LIN {X 0,Y 147.651,Z 445.005,A -85,B 0,C 180,E1 8016.217,E2 8016.217} C_VEL
LIN {X 0,Y 147.912,Z 442.573,A -85,B 0,C 180,E1 8010.384,E2 8010.384} C_VEL
LIN {X 0,Y 149.236,Z 438.224,A -85,B 0,C 180,E1 8004.615,E2 8004.615} C_VEL
LIN {X 0,Y 151.435,Z 432.256,A -85,B 0,C 180,E1 7999.344,E2 7999.344} C_VEL
LIN {X 0,Y 154.319,Z 424.793,A -85,B 0,C 180,E1 7994.592,E2 7994.592} C_VEL
LIN {X 0,Y 155.521,Z 421.178,A -85,B 0,C 180,E1 7992.697,E2 7992.697} C_VEL
LIN {X 0,Y 154.275,Z 420.555,A -85,B 0,C 180,E1 7991.775,E2 7991.775} C_VEL
LIN {X 0,Y 150.55,Z 430.544,A -85,B 0,C 180,E1 7985.489,E2 7985.489} C_VEL
LIN {X 0,Y 148.467,Z 437.566,A -85,B 0,C 180,E1 7979.547,E2 7979.547} C_VEL
LIN {X 0,Y 147.581,Z 442.658,A -85,B 0,C 180,E1 7973.399,E2 7973.399} C_VEL
LIN {X 0,Y 148.003,Z 446.153,A -85,B 0,C 180,E1 7966.855,E2 7966.855} C_VEL
LIN {X 0,Y 149.844,Z 447.721,A -85,B 0,C 180,E1 7960.472,E2 7960.472} C_VEL
LIN {X 0,Y 153.309,Z 447.472,A -85,B 0,C 180,E1 7954.074,E2 7954.074} C_VEL
LIN {X 0,Y 158.074,Z 445.504,A -85,B 0,C 180,E1 7948.321,E2 7948.321} C_VEL
LIN {X 0,Y 164.202,Z 441.703,A -85,B 0,C 180,E1 7942.937,E2 7942.937} C_VEL
LIN {X 0,Y 171.567,Z 436.08,A -85,B 0,C 180,E1 7937.992,E2 7937.992} C_VEL
LIN {X 0,Y 179.584,Z 428.799,A -85,B 0,C 180,E1 7933.693,E2 7933.693} C_VEL
LIN {X 0,Y 188.67,Z 419.109,A -85,B 0,C 180,E1 7929.691,E2 7929.691} C_VEL
LIN {X 0,Y 196.658,Z 409.241,A -85,B 0,C 180,E1 7926.716,E2 7926.716} C_VEL
LIN {X 0,Y 204.51,Z 397.865,A -85,B 0,C 180,E1 7924.143,E2 7924.143} C_VEL
LIN {X 0,Y 212.529,Z 384.144,A -85,B 0,C 180,E1 7921.803,E2 7921.803} C_VEL
LIN {X 0,Y 219.316,Z 370.142,A -85,B 0,C 180,E1 7920.001,E2 7920.001} C_VEL
LIN {X 0,Y 225.042,Z 355.307,A -85,B 0,C 180,E1 7918.566,E2 7918.566} C_VEL
LIN {X 0,Y 229.965,Z 338.612,A -85,B 0,C 180,E1 7917.371,E2 7917.371} C_VEL
LIN {X 0,Y 233.358,Z 321.906,A -85,B 0,C 180,E1 7916.537,E2 7916.537} C_VEL
LIN {X 0,Y 243.446,Z 247.809,A -85,B 0,C 180,E1 7914.255,E2 7914.255} C_VEL
LIN {X 0,Y 243.62,Z 244.534,A -85,B 0,C 180,E1 7913.875,E2 7913.875} C_VEL
LIN {X 0,Y 242.507,Z 240.131,A -85,B 0,C 180,E1 7911.703,E2 7911.703} C_VEL
LIN {X 0,Y 241.654,Z 236.36,A -85,B 0,C 180,E1 7909.149,E2 7909.149} C_VEL
LIN {X 0,Y 241.13,Z 233.586,A -85,B 0,C 180,E1 7905.594,E2 7905.594} C_VEL
LIN {X 0,Y 241.469,Z 233.295,A -85,B 0,C 180,E1 7902.157,E2 7902.157} C_VEL
LIN {X 0,Y 242.922,Z 235.401,A -85,B 0,C 180,E1 7898.258,E2 7898.258} C_VEL
LIN {X 0,Y 244.927,Z 239.89,A -85,B 0,C 180,E1 7895.046,E2 7895.046} C_VEL
LIN {X 0,Y 235.571,Z 315.768,A -85,B 0,C 180,E1 7893.078,E2 7893.078} C_VEL
LIN {X 0,Y 234.34,Z 323.435,A -85,B 0,C 180,E1 7893.125,E2 7893.125} C_VEL
LIN {X 0,Y 229.956,Z 340.511,A -85,B 0,C 180,E1 7893.896,E2 7893.896} C_VEL
LIN {X 0,Y 227.795,Z 348.034,A -85,B 0,C 180,E1 7893.937,E2 7893.937} C_VEL
LIN {X 0,Y 227.213,Z 350.101,A -85,B 0,C 180,E1 7893.868,E2 7893.868} C_VEL
LIN {X 0,Y 221.678,Z 367.592,A -85,B 0,C 180,E1 7892.977,E2 7892.977} C_VEL
LIN {X 0,Y 214.941,Z 383.787,A -85,B 0,C 180,E1 7891.828,E2 7891.828} C_VEL
LIN {X 0,Y 207.137,Z 398.997,A -85,B 0,C 180,E1 7890.33,E2 7890.33} C_VEL
LIN {X 0,Y 198.03,Z 414.01,A -85,B 0,C 180,E1 7888.297,E2 7888.297} C_VEL
LIN {X 0,Y 188.577,Z 427.423,A -85,B 0,C 180,E1 7885.805,E2 7885.805} C_VEL
LIN {X 0,Y 178.611,Z 439.75,A -85,B 0,C 180,E1 7882.65,E2 7882.65} C_VEL
LIN {X 0,Y 168.79,Z 450.698,A -85,B 0,C 180,E1 7878.794,E2 7878.794} C_VEL
LIN {X 0,Y 159.45,Z 460.267,A -85,B 0,C 180,E1 7874.113,E2 7874.113} C_VEL
LIN {X 0,Y 150.591,Z 468.9,A -85,B 0,C 180,E1 7868.135,E2 7868.135} C_VEL
LIN {X 0,Y 143.783,Z 475.492,A -85,B 0,C 180,E1 7861.439,E2 7861.439} C_VEL
LIN {X 0,Y 139.104,Z 480.495,A -85,B 0,C 180,E1 7853.739,E2 7853.739} C_VEL
LIN {X 0,Y 137.158,Z 483.651,A -85,B 0,C 180,E1 7845.651,E2 7845.651} C_VEL
LIN {X 0,Y 137.705,Z 484.936,A -85,B 0,C 180,E1 7837.933,E2 7837.933} C_VEL
LIN {X 0,Y 139.62,Z 484.587,A -85,B 0,C 180,E1 7831.234,E2 7831.234} C_VEL
LIN {X 0,Y 139.781,Z 484.641,A -85,B 0,C 180,E1 7829.593,E2 7829.593} C_VEL
LIN {X 0,Y 138.175,Z 484.8,A -85,B 0,C 180,E1 7824.189,E2 7824.189} C_VEL
LIN {X 0,Y 137.145,Z 483.177,A -85,B 0,C 180,E1 7817.666,E2 7817.666} C_VEL
LIN {X 0,Y 137.696,Z 479.482,A -85,B 0,C 180,E1 7810.931,E2 7810.931} C_VEL
LIN {X 0,Y 139.713,Z 474.37,A -85,B 0,C 180,E1 7805.028,E2 7805.028} C_VEL
LIN {X 0,Y 143.147,Z 467.343,A -85,B 0,C 180,E1 7799.347,E2 7799.347} C_VEL
LIN {X 0,Y 147.55,Z 458.752,A -85,B 0,C 180,E1 7794.359,E2 7794.359} C_VEL
LIN {X 0,Y 152.566,Z 448.608,A -85,B 0,C 180,E1 7790.045,E2 7790.045} C_VEL
LIN {X 0,Y 157.366,Z 438.016,A -85,B 0,C 180,E1 7786.675,E2 7786.675} C_VEL
LIN {X 0,Y 162.411,Z 425.199,A -85,B 0,C 180,E1 7783.646,E2 7783.646} C_VEL
LIN {X 0,Y 166.808,Z 411.49,A -85,B 0,C 180,E1 7781.293,E2 7781.293} C_VEL
LIN {X 0,Y 170.26,Z 397.535,A -85,B 0,C 180,E1 7779.582,E2 7779.582} C_VEL
LIN {X 0,Y 172.813,Z 382.764,A -85,B 0,C 180,E1 7778.363,E2 7778.363} C_VEL
LIN {X 0,Y 174.422,Z 368.061,A -85,B 0,C 180,E1 7777.585,E2 7777.585} C_VEL
LIN {X 0,Y 177.852,Z 350.466,A -85,B 0,C 180,E1 7776.2,E2 7776.2} C_VEL
LIN {X 0,Y 180.054,Z 332.064,A -85,B 0,C 180,E1 7775.237,E2 7775.237} C_VEL
LIN {X 0,Y 188.013,Z 232.01,A -85,B 0,C 180,E1 7771.757,E2 7771.757} C_VEL
LIN {X 0,Y 195.653,Z 198.676,A -85,B 0,C 180,E1 7769.476,E2 7769.476} C_VEL
LIN {X 0,Y 193.33,Z 185.485,A -85,B 0,C 180,E1 7765.092,E2 7765.092} C_VEL
LIN {X 0,Y 191.37,Z 173.485,A -85,B 0,C 180,E1 7760.171,E2 7760.171} C_VEL
LIN {X 0,Y 190.931,Z 170.626,A -85,B 0,C 180,E1 7758.629,E2 7758.629} C_VEL
LIN {X 0,Y 189.927,Z 168.519,A -85,B 0,C 180,E1 7756.515,E2 7756.515} C_VEL
LIN {X 0,Y 186.759,Z 164.115,A -85,B 0,C 180,E1 7747.382,E2 7747.382} C_VEL
LIN {X 0,Y 186.26,Z 164.227,A -85,B 0,C 180,E1 7743.693,E2 7743.693} C_VEL
LIN {X 0,Y 186.938,Z 167.789,A -85,B 0,C 180,E1 7734.782,E2 7734.782} C_VEL
LIN {X 0,Y 188.283,Z 172.083,A -85,B 0,C 180,E1 7729.906,E2 7729.906} C_VEL
LIN {X 0,Y 189.759,Z 176.341,A -85,B 0,C 180,E1 7726.283,E2 7726.283} C_VEL
LIN {X 0,Y 191.495,Z 181.495,A -85,B 0,C 180,E1 7722.685,E2 7722.685} C_VEL
LIN {X 0,Y 193.745,Z 189.705,A -85,B 0,C 180,E1 7718.187,E2 7718.187} C_VEL
LIN {X 0,Y 195.931,Z 198.744,A -85,B 0,C 180,E1 7714.293,E2 7714.293} C_VEL
LIN {X 0,Y 197.495,Z 207.805,A -85,B 0,C 180,E1 7711.044,E2 7711.044} C_VEL
LIN {X 0,Y 193.191,Z 231.562,A -85,B 0,C 180,E1 7707.459,E2 7707.459} C_VEL
LIN {X 0,Y 193.556,Z 239.75,A -85,B 0,C 180,E1 7706.786,E2 7706.786} C_VEL
LIN {X 0,Y 187.438,Z 320.364,A -85,B 0,C 180,E1 7704.244,E2 7704.244} C_VEL
LIN {X 0,Y 185.829,Z 348.64,A -85,B 0,C 180,E1 7702.979,E2 7702.979} C_VEL
